// Mitsubishi GX Developer project: 12-202_201204121600   PLC: FX3U

PROGRAM MAIN
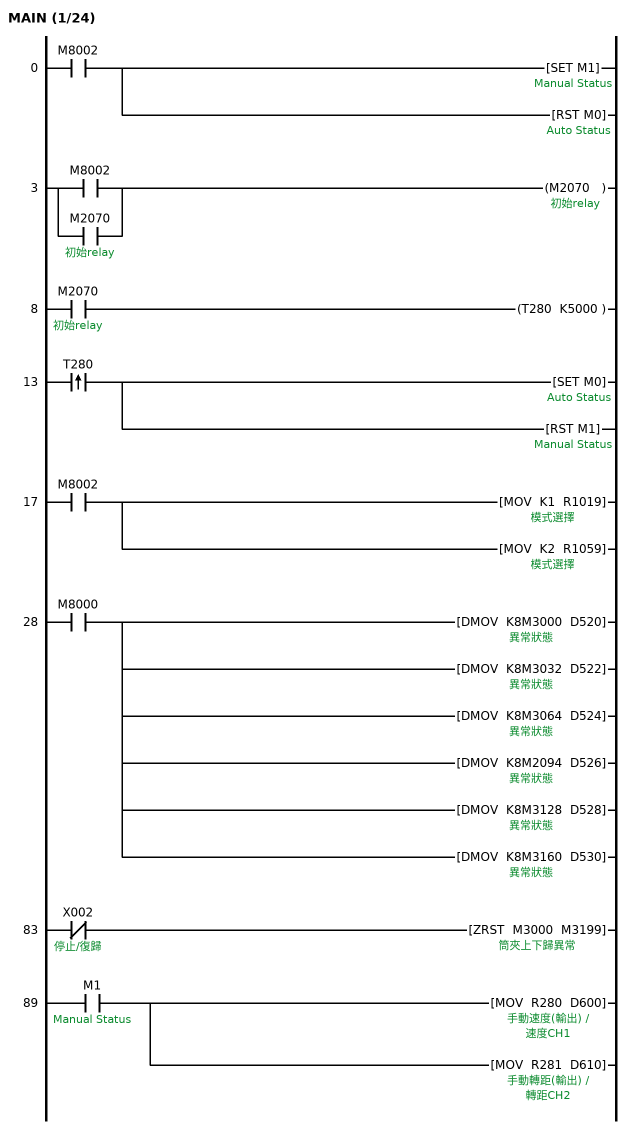
0     LD      M8002
      SET     M1  ; Manual Status
      RST     M0  ; Auto Status
3     LD      M8002
      OR      M2070  ; 初始relay
      OUT     M2070  ; 初始relay
8     LD      M2070  ; 初始relay
      OUT     T280 K5000
13    LDP     T280
      SET     M0  ; Auto Status
      RST     M1  ; Manual Status
17    LD      M8002
      MOV     K1 R1019  ; 模式選擇
      MOV     K2 R1059  ; 模式選擇
28    LD      M8000
      DMOV    K8M3000 D520  ; 筒夾上下歸異常 / 異常狀態
      DMOV    K8M3032 D522  ; 異常狀態
      DMOV    K8M3064 D524  ; 異常狀態
      DMOV    K8M2094 D526  ; 異常狀態
      DMOV    K8M3128 D528  ; 異常狀態
      DMOV    K8M3160 D530  ; 異常狀態
83    LDI     X002  ; 停止/復歸
      ZRST    M3000 M3199
89    LD      M1  ; Manual Status
      MOV     R280 D600  ; 手動速度(輸出) / 速度CH1
      MOV     R281 D610  ; 手動轉距(輸出) / 轉距CH2
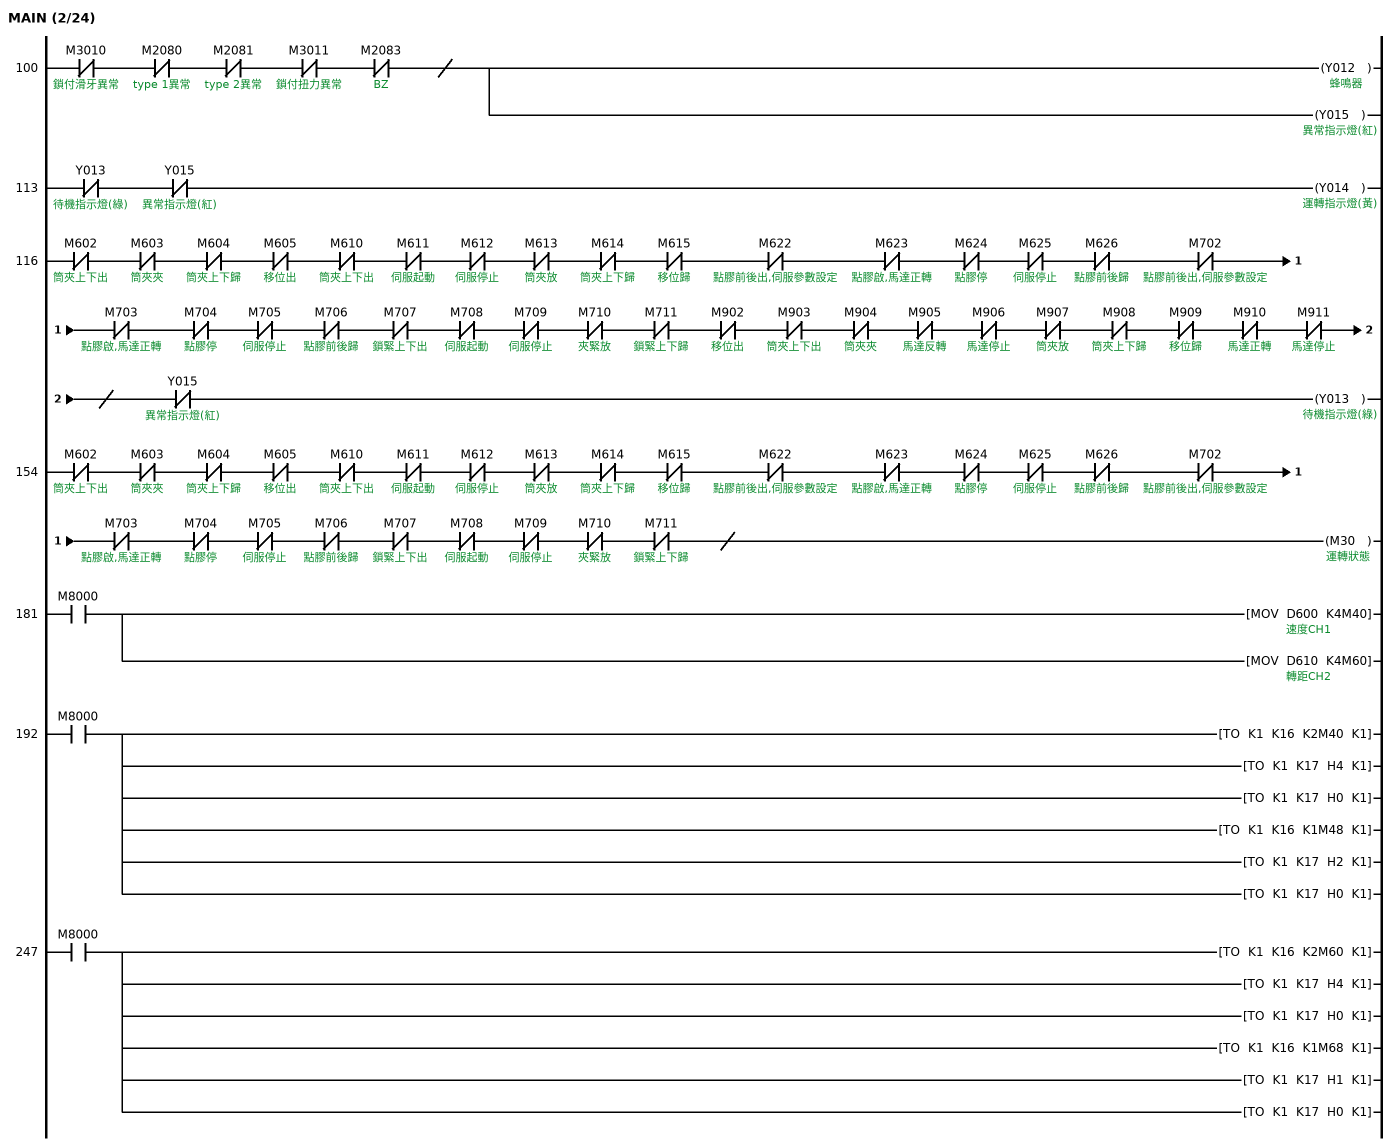
100   LDI     M3010  ; 鎖付滑牙異常
      ANI     M2080  ; type 1異常
      ANI     M2081  ; type 2異常
      ANI     M3011  ; 鎖付扭力異常
      ANI     M2083  ; BZ
      INV
      OUT     Y012  ; 蜂鳴器
      OUT     Y015  ; 異常指示燈(紅)
113   LDI     Y013  ; 待機指示燈(綠)
      ANI     Y015  ; 異常指示燈(紅)
      OUT     Y014  ; 運轉指示燈(黃)
116   LDI     M602  ; 筒夾上下出
      ANI     M603  ; 筒夾夾
      ANI     M604  ; 筒夾上下歸
      ANI     M605  ; 移位出
      ANI     M610  ; 筒夾上下出
      ANI     M611  ; 伺服起動
      ANI     M612  ; 伺服停止
      ANI     M613  ; 筒夾放
      ANI     M614  ; 筒夾上下歸
      ANI     M615  ; 移位歸
      ANI     M622  ; 點膠前後出,伺服參數設定
      ANI     M623  ; 點膠啟,馬達正轉
      ANI     M624  ; 點膠停
      ANI     M625  ; 伺服停止
      ANI     M626  ; 點膠前後歸
      ANI     M702  ; 點膠前後出,伺服參數設定
      ANI     M703  ; 點膠啟,馬達正轉
      ANI     M704  ; 點膠停
      ANI     M705  ; 伺服停止
      ANI     M706  ; 點膠前後歸
      ANI     M707  ; 鎖緊上下出
      ANI     M708  ; 伺服起動
      ANI     M709  ; 伺服停止
      ANI     M710  ; 夾緊放
      ANI     M711  ; 鎖緊上下歸
      ANI     M902  ; 移位出
      ANI     M903  ; 筒夾上下出
      ANI     M904  ; 筒夾夾
      ANI     M905  ; 馬達反轉
      ANI     M906  ; 馬達停止
      ANI     M907  ; 筒夾放
      ANI     M908  ; 筒夾上下歸
      ANI     M909  ; 移位歸
      ANI     M910  ; 馬達正轉
      ANI     M911  ; 馬達停止
      INV
      ANI     Y015  ; 異常指示燈(紅)
      OUT     Y013  ; 待機指示燈(綠)
154   LDI     M602  ; 筒夾上下出
      ANI     M603  ; 筒夾夾
      ANI     M604  ; 筒夾上下歸
      ANI     M605  ; 移位出
      ANI     M610  ; 筒夾上下出
      ANI     M611  ; 伺服起動
      ANI     M612  ; 伺服停止
      ANI     M613  ; 筒夾放
      ANI     M614  ; 筒夾上下歸
      ANI     M615  ; 移位歸
      ANI     M622  ; 點膠前後出,伺服參數設定
      ANI     M623  ; 點膠啟,馬達正轉
      ANI     M624  ; 點膠停
      ANI     M625  ; 伺服停止
      ANI     M626  ; 點膠前後歸
      ANI     M702  ; 點膠前後出,伺服參數設定
      ANI     M703  ; 點膠啟,馬達正轉
      ANI     M704  ; 點膠停
      ANI     M705  ; 伺服停止
      ANI     M706  ; 點膠前後歸
      ANI     M707  ; 鎖緊上下出
      ANI     M708  ; 伺服起動
      ANI     M709  ; 伺服停止
      ANI     M710  ; 夾緊放
      ANI     M711  ; 鎖緊上下歸
      INV
      OUT     M30  ; 運轉狀態
181   LD      M8000
      MOV     D600 K4M40  ; DA用
      MOV     D610 K4M60  ; DA用
192   LD      M8000
      TO      K1 K16 K2M40 K1
      TO      K1 K17 H4 K1
      TO      K1 K17 H0 K1
      TO      K1 K16 K1M48 K1  ; DA用
      TO      K1 K17 H2 K1
      TO      K1 K17 H0 K1
247   LD      M8000
      TO      K1 K16 K2M60 K1
      TO      K1 K17 H4 K1
      TO      K1 K17 H0 K1
      TO      K1 K16 K1M68 K1  ; DA用
      TO      K1 K17 H1 K1
      TO      K1 K17 H0 K1
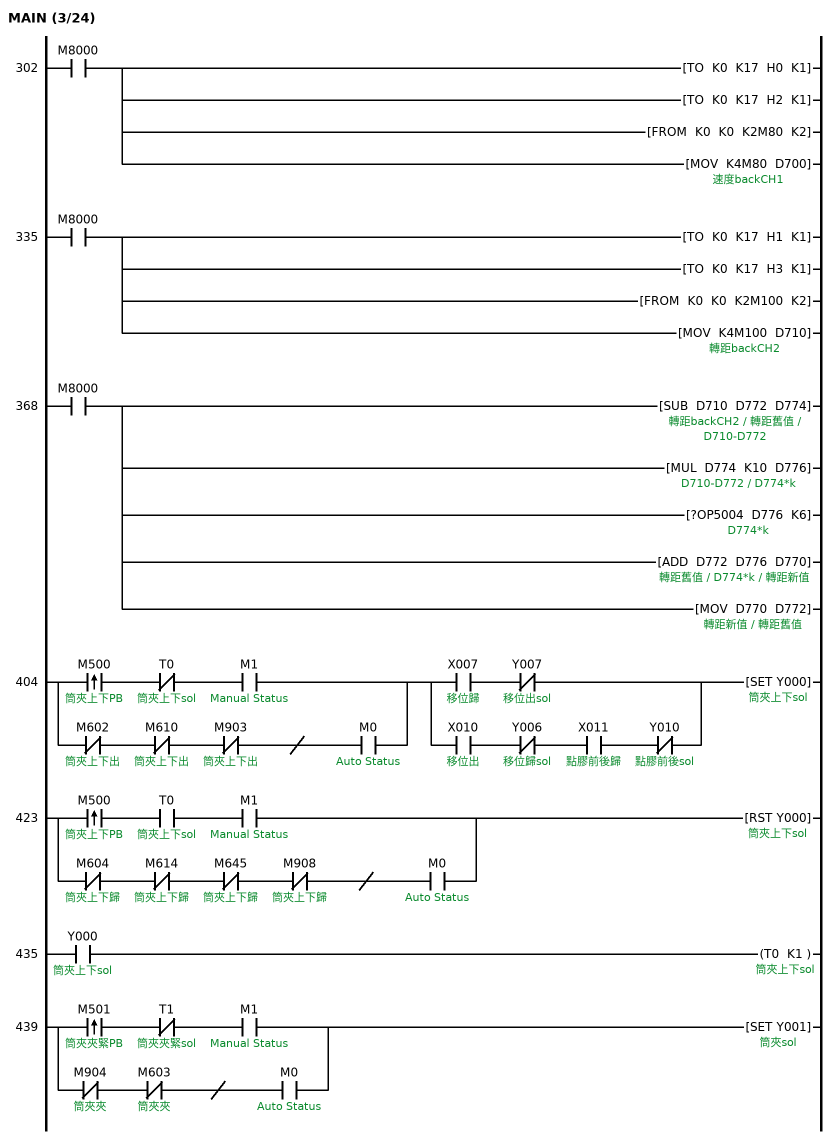
302   LD      M8000
      TO      K0 K17 H0 K1
      TO      K0 K17 H2 K1
      FROM    K0 K0 K2M80 K2  ; AD用
      MOV     K4M80 D700  ; 速度backCH1
335   LD      M8000
      TO      K0 K17 H1 K1
      TO      K0 K17 H3 K1
      FROM    K0 K0 K2M100 K2  ; AD用
      MOV     K4M100 D710  ; 轉距backCH2
368   LD      M8000
      SUB     D710 D772 D774  ; 轉距舊值 / D710-D772
      MUL     D774 K10 D776  ; D774*k
      ?OP5004 D776 K6
      ADD     D772 D776 D770  ; 轉距新值
      MOV     D770 D772
404   LDP     M500  ; 筒夾上下PB
      ANI     T0  ; 筒夾上下sol
      AND     M1  ; Manual Status
      LDI     M602  ; 筒夾上下出
      ANI     M610  ; 筒夾上下出
      ANI     M903  ; 筒夾上下出
      INV
      AND     M0  ; Auto Status
      ORB
      LD      X007  ; 移位歸
      ANI     Y007  ; 移位出sol
      LD      X010  ; 移位出
      ANI     Y006  ; 移位歸sol
      AND     X011  ; 點膠前後歸
      ANI     Y010  ; 點膠前後sol
      ORB
      ANB
      SET     Y000  ; 筒夾上下sol
423   LDP     M500  ; 筒夾上下PB
      AND     T0  ; 筒夾上下sol
      AND     M1  ; Manual Status
      LDI     M604  ; 筒夾上下歸
      ANI     M614  ; 筒夾上下歸
      ANI     M645  ; 筒夾上下歸
      ANI     M908  ; 筒夾上下歸
      INV
      AND     M0  ; Auto Status
      ORB
      RST     Y000  ; 筒夾上下sol
435   LD      Y000  ; 筒夾上下sol
      OUT     T0 K1  ; 筒夾上下sol
439   LDP     M501  ; 筒夾夾緊PB
      ANI     T1  ; 筒夾夾緊sol
      AND     M1  ; Manual Status
      LDI     M904  ; 筒夾夾
      ANI     M603  ; 筒夾夾
      INV
      AND     M0  ; Auto Status
      ORB
      SET     Y001  ; 筒夾sol
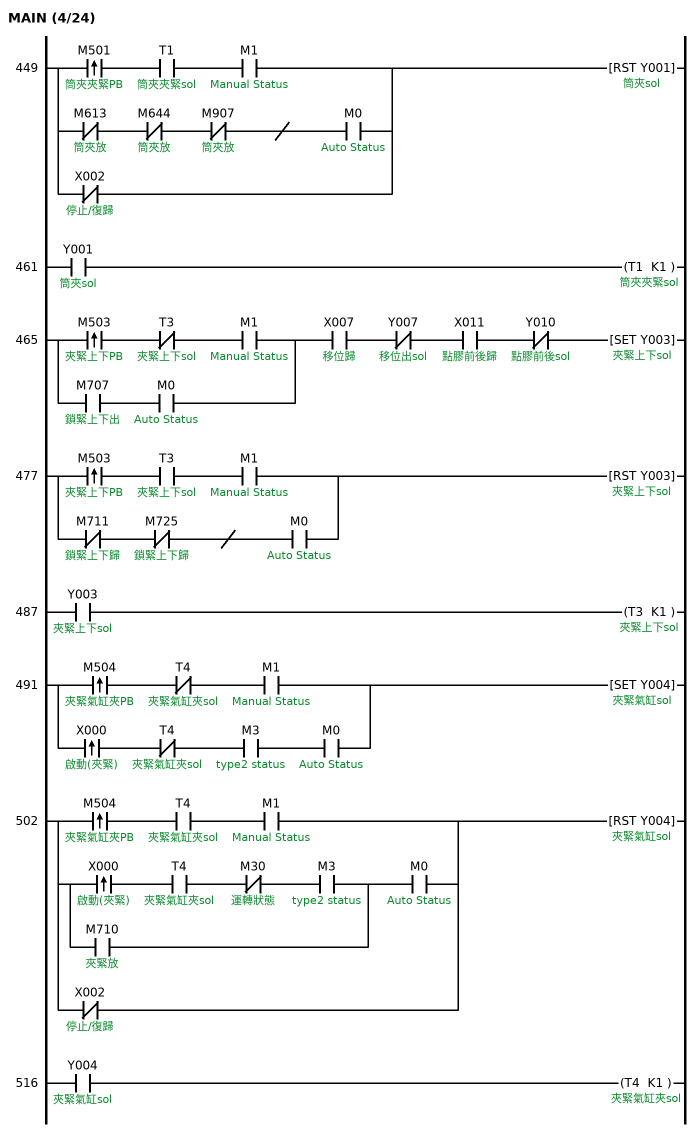
449   LDP     M501  ; 筒夾夾緊PB
      AND     T1  ; 筒夾夾緊sol
      AND     M1  ; Manual Status
      LDI     M613  ; 筒夾放
      ANI     M644  ; 筒夾放
      ANI     M907  ; 筒夾放
      INV
      AND     M0  ; Auto Status
      ORB
      ORI     X002  ; 停止/復歸
      RST     Y001  ; 筒夾sol
461   LD      Y001  ; 筒夾sol
      OUT     T1 K1  ; 筒夾夾緊sol
465   LDP     M503  ; 夾緊上下PB
      ANI     T3  ; 夾緊上下sol
      AND     M1  ; Manual Status
      LD      M707  ; 鎖緊上下出
      AND     M0  ; Auto Status
      ORB
      AND     X007  ; 移位歸
      ANI     Y007  ; 移位出sol
      AND     X011  ; 點膠前後歸
      ANI     Y010  ; 點膠前後sol
      SET     Y003  ; 夾緊上下sol
477   LDP     M503  ; 夾緊上下PB
      AND     T3  ; 夾緊上下sol
      AND     M1  ; Manual Status
      LDI     M711  ; 鎖緊上下歸
      ANI     M725  ; 鎖緊上下歸
      INV
      AND     M0  ; Auto Status
      ORB
      RST     Y003  ; 夾緊上下sol
487   LD      Y003  ; 夾緊上下sol
      OUT     T3 K1  ; 夾緊上下sol
491   LDP     M504  ; 夾緊氣缸夾PB
      ANI     T4  ; 夾緊氣缸夾sol
      AND     M1  ; Manual Status
      LDP     X000  ; 啟動(夾緊)
      ANI     T4  ; 夾緊氣缸夾sol
      AND     M3  ; type2 status
      AND     M0  ; Auto Status
      ORB
      SET     Y004  ; 夾緊氣缸sol
502   LDP     M504  ; 夾緊氣缸夾PB
      AND     T4  ; 夾緊氣缸夾sol
      AND     M1  ; Manual Status
      LDP     X000  ; 啟動(夾緊)
      AND     T4  ; 夾緊氣缸夾sol
      ANI     M30  ; 運轉狀態
      AND     M3  ; type2 status
      OR      M710  ; 夾緊放
      AND     M0  ; Auto Status
      ORB
      ORI     X002  ; 停止/復歸
      RST     Y004  ; 夾緊氣缸sol
516   LD      Y004  ; 夾緊氣缸sol
      OUT     T4 K1  ; 夾緊氣缸夾sol
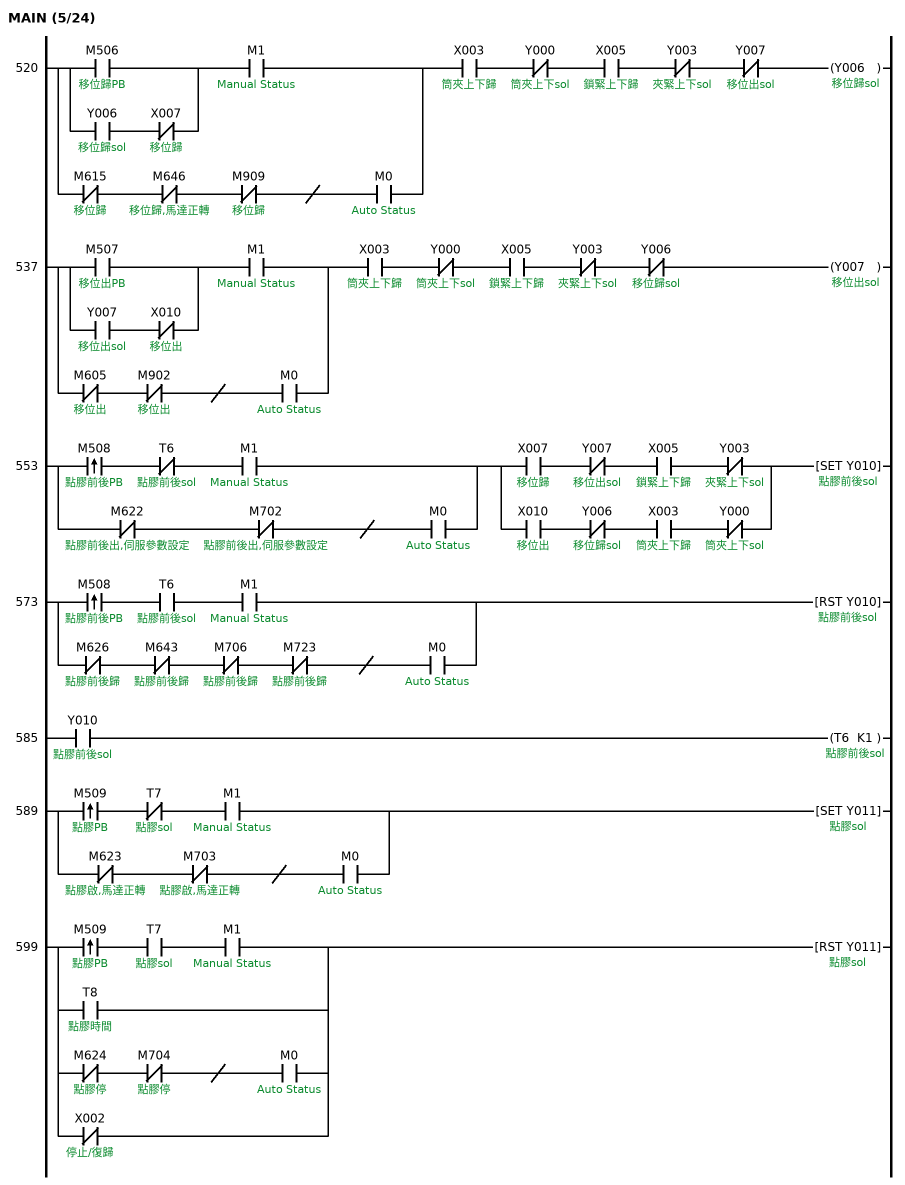
520   LD      M506  ; 移位歸PB
      LD      Y006  ; 移位歸sol
      ANI     X007  ; 移位歸
      ORB
      AND     M1  ; Manual Status
      LDI     M615  ; 移位歸
      ANI     M646  ; 移位歸,馬達正轉
      ANI     M909  ; 移位歸
      INV
      AND     M0  ; Auto Status
      ORB
      AND     X003  ; 筒夾上下歸
      ANI     Y000  ; 筒夾上下sol
      AND     X005  ; 鎖緊上下歸
      ANI     Y003  ; 夾緊上下sol
      ANI     Y007  ; 移位出sol
      OUT     Y006  ; 移位歸sol
537   LD      M507  ; 移位出PB
      LD      Y007  ; 移位出sol
      ANI     X010  ; 移位出
      ORB
      AND     M1  ; Manual Status
      LDI     M605  ; 移位出
      ANI     M902  ; 移位出
      INV
      AND     M0  ; Auto Status
      ORB
      AND     X003  ; 筒夾上下歸
      ANI     Y000  ; 筒夾上下sol
      AND     X005  ; 鎖緊上下歸
      ANI     Y003  ; 夾緊上下sol
      ANI     Y006  ; 移位歸sol
      OUT     Y007  ; 移位出sol
553   LDP     M508  ; 點膠前後PB
      ANI     T6  ; 點膠前後sol
      AND     M1  ; Manual Status
      LDI     M622  ; 點膠前後出,伺服參數設定
      ANI     M702  ; 點膠前後出,伺服參數設定
      INV
      AND     M0  ; Auto Status
      ORB
      LD      X007  ; 移位歸
      ANI     Y007  ; 移位出sol
      AND     X005  ; 鎖緊上下歸
      ANI     Y003  ; 夾緊上下sol
      LD      X010  ; 移位出
      ANI     Y006  ; 移位歸sol
      AND     X003  ; 筒夾上下歸
      ANI     Y000  ; 筒夾上下sol
      ORB
      ANB
      SET     Y010  ; 點膠前後sol
573   LDP     M508  ; 點膠前後PB
      AND     T6  ; 點膠前後sol
      AND     M1  ; Manual Status
      LDI     M626  ; 點膠前後歸
      ANI     M643  ; 點膠前後歸
      ANI     M706  ; 點膠前後歸
      ANI     M723  ; 點膠前後歸
      INV
      AND     M0  ; Auto Status
      ORB
      RST     Y010  ; 點膠前後sol
585   LD      Y010  ; 點膠前後sol
      OUT     T6 K1  ; 點膠前後sol
589   LDP     M509  ; 點膠PB
      ANI     T7  ; 點膠sol
      AND     M1  ; Manual Status
      LDI     M623  ; 點膠啟,馬達正轉
      ANI     M703  ; 點膠啟,馬達正轉
      INV
      AND     M0  ; Auto Status
      ORB
      SET     Y011  ; 點膠sol
599   LDP     M509  ; 點膠PB
      AND     T7  ; 點膠sol
      AND     M1  ; Manual Status
      OR      T8  ; 點膠時間
      LDI     M624  ; 點膠停
      ANI     M704  ; 點膠停
      INV
      AND     M0  ; Auto Status
      ORB
      ORI     X002  ; 停止/復歸
      RST     Y011  ; 點膠sol
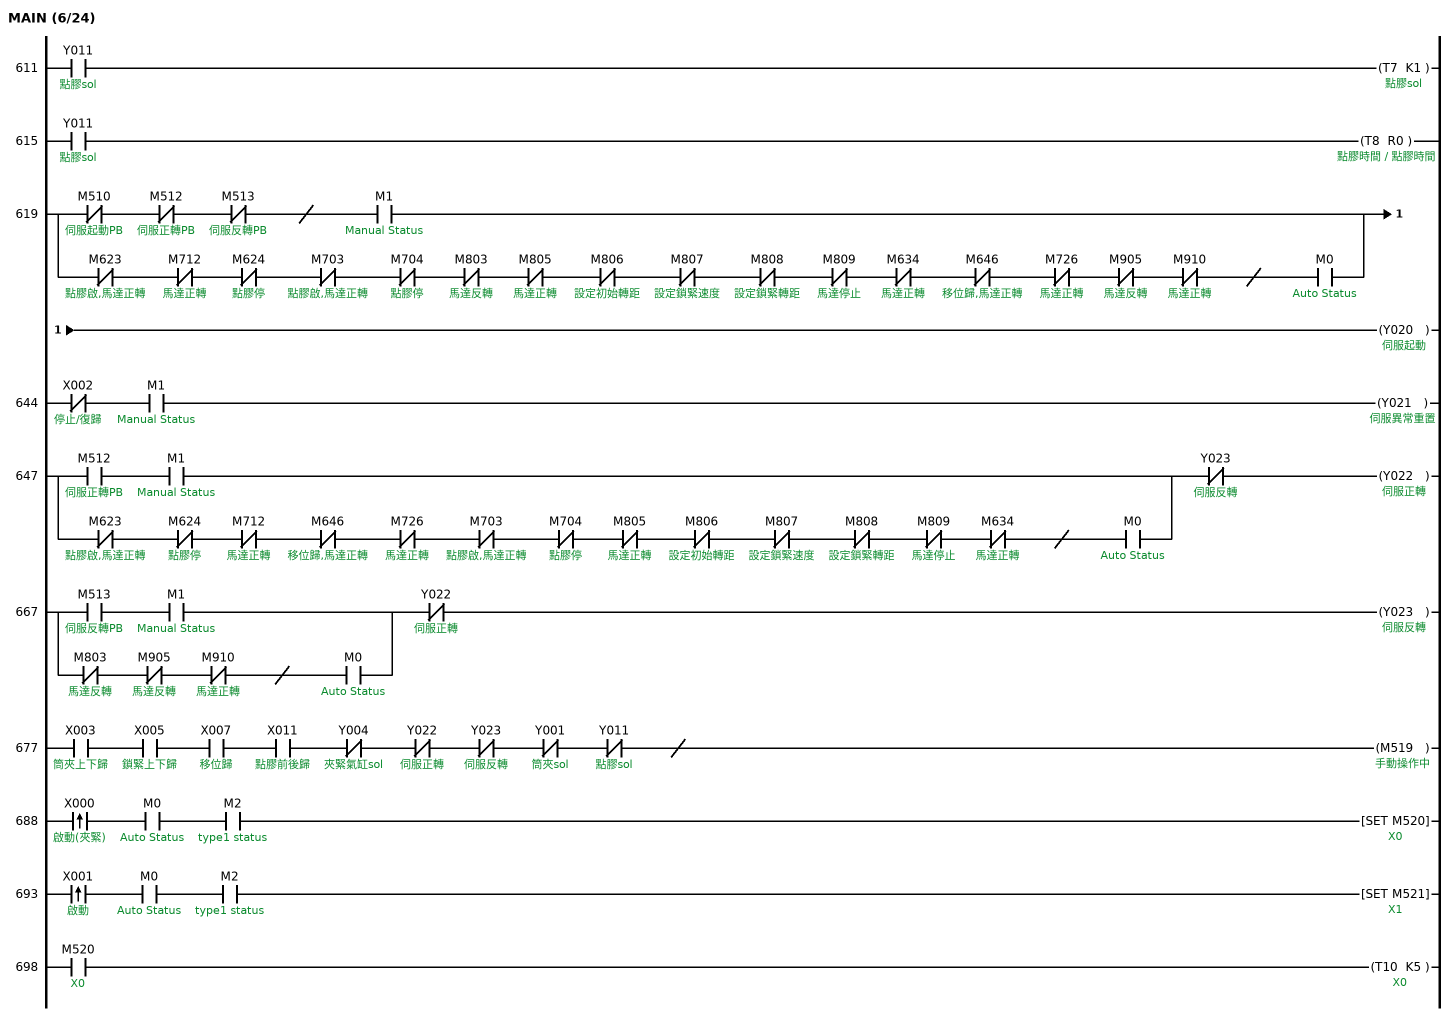
611   LD      Y011  ; 點膠sol
      OUT     T7 K1  ; 點膠sol
615   LD      Y011  ; 點膠sol
      OUT     T8 R0  ; 點膠時間 / 點膠時間
619   LDI     M510  ; 伺服起動PB
      ANI     M512  ; 伺服正轉PB
      ANI     M513  ; 伺服反轉PB
      INV
      AND     M1  ; Manual Status
      LDI     M623  ; 點膠啟,馬達正轉
      ANI     M712  ; 馬達正轉
      ANI     M624  ; 點膠停
      ANI     M703  ; 點膠啟,馬達正轉
      ANI     M704  ; 點膠停
      ANI     M803  ; 馬達反轉
      ANI     M805  ; 馬達正轉
      ANI     M806  ; 設定初始轉距
      ANI     M807  ; 設定鎖緊速度
      ANI     M808  ; 設定鎖緊轉距
      ANI     M809  ; 馬達停止
      ANI     M634  ; 馬達正轉
      ANI     M646  ; 移位歸,馬達正轉
      ANI     M726  ; 馬達正轉
      ANI     M905  ; 馬達反轉
      ANI     M910  ; 馬達正轉
      INV
      AND     M0  ; Auto Status
      ORB
      OUT     Y020  ; 伺服起動
644   LDI     X002  ; 停止/復歸
      AND     M1  ; Manual Status
      OUT     Y021  ; 伺服異常重置
647   LD      M512  ; 伺服正轉PB
      AND     M1  ; Manual Status
      LDI     M623  ; 點膠啟,馬達正轉
      ANI     M624  ; 點膠停
      ANI     M712  ; 馬達正轉
      ANI     M646  ; 移位歸,馬達正轉
      ANI     M726  ; 馬達正轉
      ANI     M703  ; 點膠啟,馬達正轉
      ANI     M704  ; 點膠停
      ANI     M805  ; 馬達正轉
      ANI     M806  ; 設定初始轉距
      ANI     M807  ; 設定鎖緊速度
      ANI     M808  ; 設定鎖緊轉距
      ANI     M809  ; 馬達停止
      ANI     M634  ; 馬達正轉
      INV
      AND     M0  ; Auto Status
      ORB
      ANI     Y023  ; 伺服反轉
      OUT     Y022  ; 伺服正轉
667   LD      M513  ; 伺服反轉PB
      AND     M1  ; Manual Status
      LDI     M803  ; 馬達反轉
      ANI     M905  ; 馬達反轉
      ANI     M910  ; 馬達正轉
      INV
      AND     M0  ; Auto Status
      ORB
      ANI     Y022  ; 伺服正轉
      OUT     Y023  ; 伺服反轉
677   LD      X003  ; 筒夾上下歸
      AND     X005  ; 鎖緊上下歸
      AND     X007  ; 移位歸
      AND     X011  ; 點膠前後歸
      ANI     Y004  ; 夾緊氣缸sol
      ANI     Y022  ; 伺服正轉
      ANI     Y023  ; 伺服反轉
      ANI     Y001  ; 筒夾sol
      ANI     Y011  ; 點膠sol
      INV
      OUT     M519  ; 手動操作中
688   LDP     X000  ; 啟動(夾緊)
      AND     M0  ; Auto Status
      AND     M2  ; type1 status
      SET     M520  ; X0
693   LDP     X001  ; 啟動
      AND     M0  ; Auto Status
      AND     M2  ; type1 status
      SET     M521  ; X1
698   LD      M520  ; X0
      OUT     T10 K5  ; X0
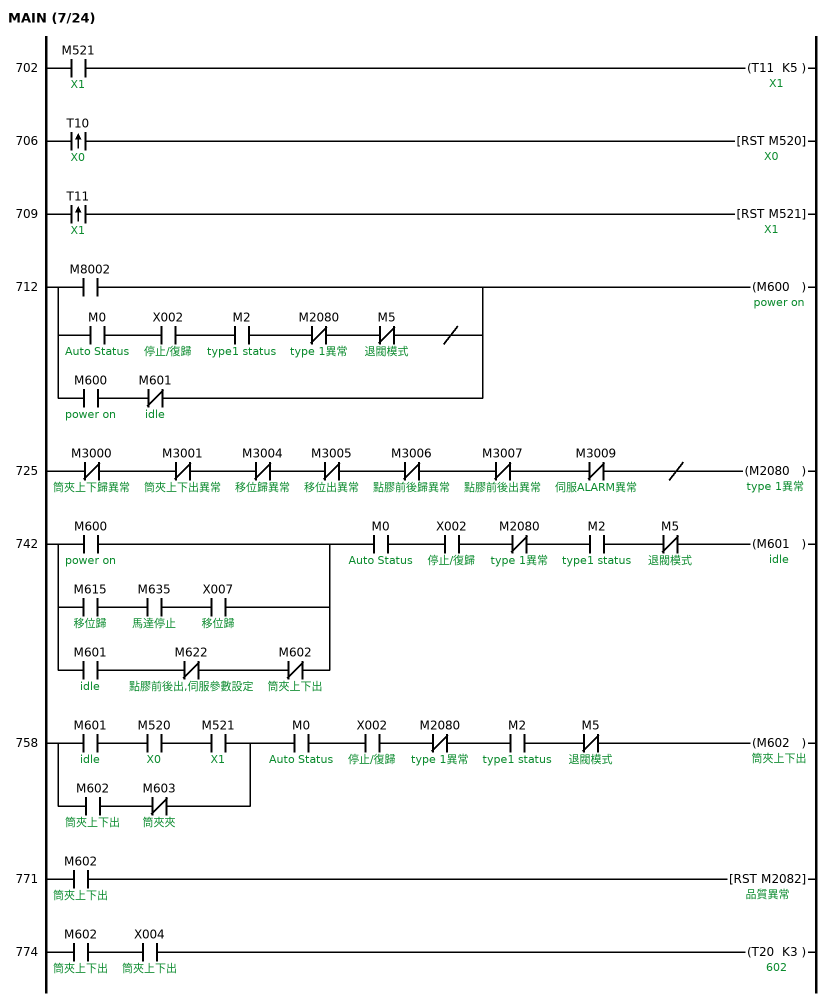
702   LD      M521  ; X1
      OUT     T11 K5  ; X1
706   LDP     T10  ; X0
      RST     M520  ; X0
709   LDP     T11  ; X1
      RST     M521  ; X1
712   LD      M8002
      LD      M0  ; Auto Status
      AND     X002  ; 停止/復歸
      AND     M2  ; type1 status
      ANI     M2080  ; type 1異常
      ANI     M5  ; 退閥模式
      INV
      ORB
      LD      M600  ; power on
      ANI     M601  ; idle
      ORB
      OUT     M600  ; power on
725   LDI     M3000  ; 筒夾上下歸異常
      ANI     M3001  ; 筒夾上下出異常
      ANI     M3004  ; 移位歸異常
      ANI     M3005  ; 移位出異常
      ANI     M3006  ; 點膠前後歸異常
      ANI     M3007  ; 點膠前後出異常
      ANI     M3009  ; 伺服ALARM異常
      INV
      OUT     M2080  ; type 1異常
742   LD      M600  ; power on
      LD      M615  ; 移位歸
      AND     M635  ; 馬達停止
      AND     X007  ; 移位歸
      ORB
      LD      M601  ; idle
      ANI     M622  ; 點膠前後出,伺服參數設定
      ANI     M602  ; 筒夾上下出
      ORB
      AND     M0  ; Auto Status
      AND     X002  ; 停止/復歸
      ANI     M2080  ; type 1異常
      AND     M2  ; type1 status
      ANI     M5  ; 退閥模式
      OUT     M601  ; idle
758   LD      M601  ; idle
      AND     M520  ; X0
      AND     M521  ; X1
      LD      M602  ; 筒夾上下出
      ANI     M603  ; 筒夾夾
      ORB
      AND     M0  ; Auto Status
      AND     X002  ; 停止/復歸
      ANI     M2080  ; type 1異常
      AND     M2  ; type1 status
      ANI     M5  ; 退閥模式
      OUT     M602  ; 筒夾上下出
771   LD      M602  ; 筒夾上下出
      RST     M2082  ; 品質異常
774   LD      M602  ; 筒夾上下出
      AND     X004  ; 筒夾上下出
      OUT     T20 K3  ; 602
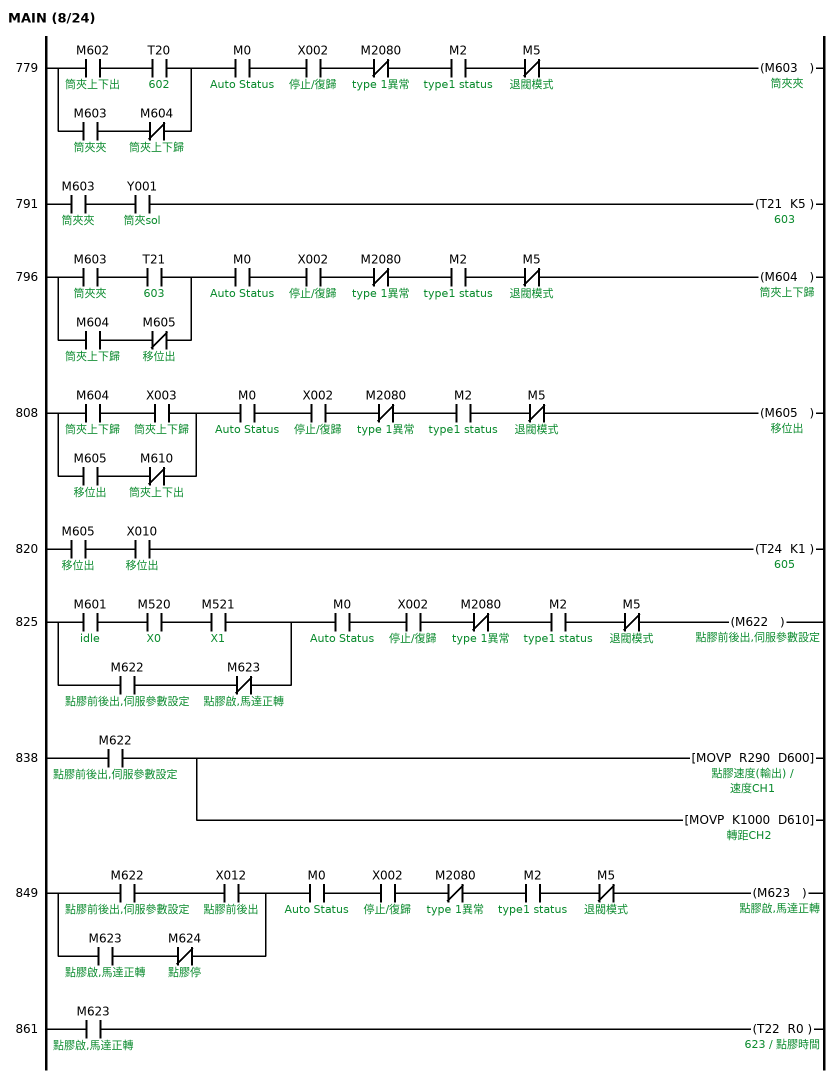
779   LD      M602  ; 筒夾上下出
      AND     T20  ; 602
      LD      M603  ; 筒夾夾
      ANI     M604  ; 筒夾上下歸
      ORB
      AND     M0  ; Auto Status
      AND     X002  ; 停止/復歸
      ANI     M2080  ; type 1異常
      AND     M2  ; type1 status
      ANI     M5  ; 退閥模式
      OUT     M603  ; 筒夾夾
791   LD      M603  ; 筒夾夾
      AND     Y001  ; 筒夾sol
      OUT     T21 K5  ; 603
796   LD      M603  ; 筒夾夾
      AND     T21  ; 603
      LD      M604  ; 筒夾上下歸
      ANI     M605  ; 移位出
      ORB
      AND     M0  ; Auto Status
      AND     X002  ; 停止/復歸
      ANI     M2080  ; type 1異常
      AND     M2  ; type1 status
      ANI     M5  ; 退閥模式
      OUT     M604  ; 筒夾上下歸
808   LD      M604  ; 筒夾上下歸
      AND     X003  ; 筒夾上下歸
      LD      M605  ; 移位出
      ANI     M610  ; 筒夾上下出
      ORB
      AND     M0  ; Auto Status
      AND     X002  ; 停止/復歸
      ANI     M2080  ; type 1異常
      AND     M2  ; type1 status
      ANI     M5  ; 退閥模式
      OUT     M605  ; 移位出
820   LD      M605  ; 移位出
      AND     X010  ; 移位出
      OUT     T24 K1  ; 605
825   LD      M601  ; idle
      AND     M520  ; X0
      AND     M521  ; X1
      LD      M622  ; 點膠前後出,伺服參數設定
      ANI     M623  ; 點膠啟,馬達正轉
      ORB
      AND     M0  ; Auto Status
      AND     X002  ; 停止/復歸
      ANI     M2080  ; type 1異常
      AND     M2  ; type1 status
      ANI     M5  ; 退閥模式
      OUT     M622  ; 點膠前後出,伺服參數設定
838   LD      M622  ; 點膠前後出,伺服參數設定
      MOVP    R290 D600  ; 點膠速度(輸出)
      MOVP    K1000 D610
849   LD      M622  ; 點膠前後出,伺服參數設定
      AND     X012  ; 點膠前後出
      LD      M623  ; 點膠啟,馬達正轉
      ANI     M624  ; 點膠停
      ORB
      AND     M0  ; Auto Status
      AND     X002  ; 停止/復歸
      ANI     M2080  ; type 1異常
      AND     M2  ; type1 status
      ANI     M5  ; 退閥模式
      OUT     M623  ; 點膠啟,馬達正轉
861   LD      M623  ; 點膠啟,馬達正轉
      OUT     T22 R0  ; 623 / 點膠時間
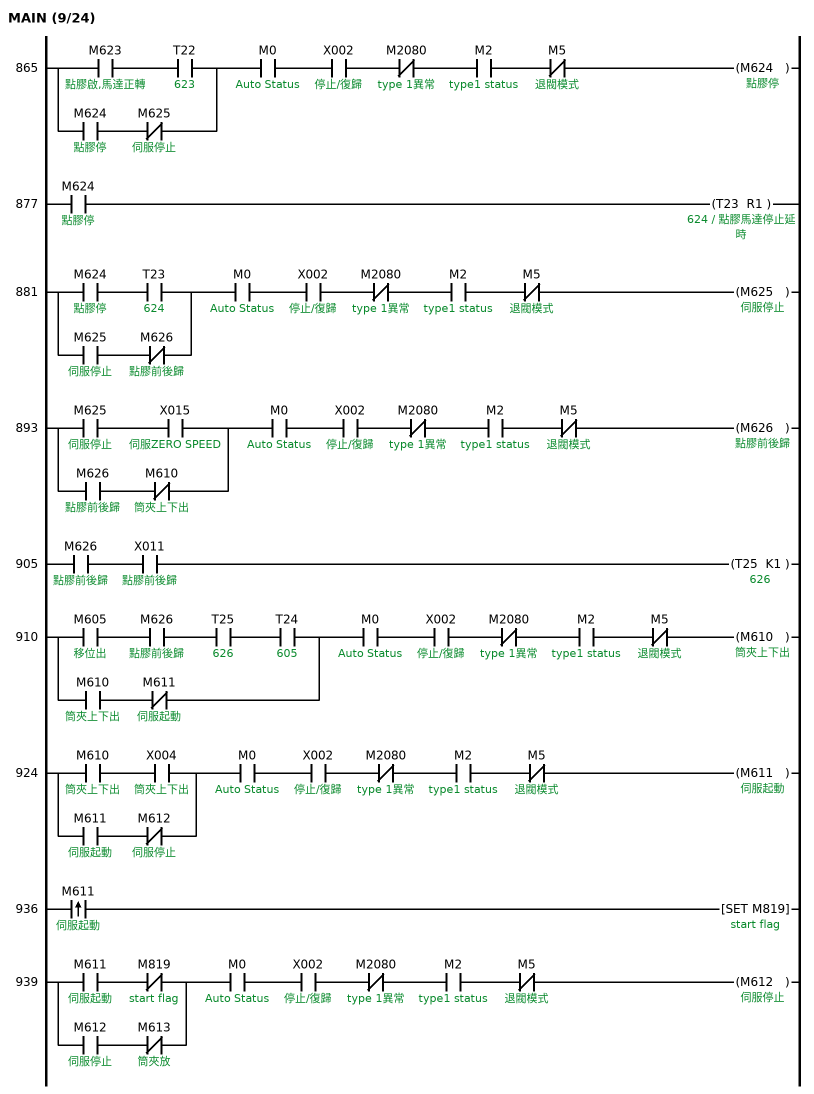
865   LD      M623  ; 點膠啟,馬達正轉
      AND     T22  ; 623
      LD      M624  ; 點膠停
      ANI     M625  ; 伺服停止
      ORB
      AND     M0  ; Auto Status
      AND     X002  ; 停止/復歸
      ANI     M2080  ; type 1異常
      AND     M2  ; type1 status
      ANI     M5  ; 退閥模式
      OUT     M624  ; 點膠停
877   LD      M624  ; 點膠停
      OUT     T23 R1  ; 624 / 點膠馬達停止延時
881   LD      M624  ; 點膠停
      AND     T23  ; 624
      LD      M625  ; 伺服停止
      ANI     M626  ; 點膠前後歸
      ORB
      AND     M0  ; Auto Status
      AND     X002  ; 停止/復歸
      ANI     M2080  ; type 1異常
      AND     M2  ; type1 status
      ANI     M5  ; 退閥模式
      OUT     M625  ; 伺服停止
893   LD      M625  ; 伺服停止
      AND     X015  ; 伺服ZERO SPEED
      LD      M626  ; 點膠前後歸
      ANI     M610  ; 筒夾上下出
      ORB
      AND     M0  ; Auto Status
      AND     X002  ; 停止/復歸
      ANI     M2080  ; type 1異常
      AND     M2  ; type1 status
      ANI     M5  ; 退閥模式
      OUT     M626  ; 點膠前後歸
905   LD      M626  ; 點膠前後歸
      AND     X011  ; 點膠前後歸
      OUT     T25 K1  ; 626
910   LD      M605  ; 移位出
      AND     M626  ; 點膠前後歸
      AND     T25  ; 626
      AND     T24  ; 605
      LD      M610  ; 筒夾上下出
      ANI     M611  ; 伺服起動
      ORB
      AND     M0  ; Auto Status
      AND     X002  ; 停止/復歸
      ANI     M2080  ; type 1異常
      AND     M2  ; type1 status
      ANI     M5  ; 退閥模式
      OUT     M610  ; 筒夾上下出
924   LD      M610  ; 筒夾上下出
      AND     X004  ; 筒夾上下出
      LD      M611  ; 伺服起動
      ANI     M612  ; 伺服停止
      ORB
      AND     M0  ; Auto Status
      AND     X002  ; 停止/復歸
      ANI     M2080  ; type 1異常
      AND     M2  ; type1 status
      ANI     M5  ; 退閥模式
      OUT     M611  ; 伺服起動
936   LDP     M611  ; 伺服起動
      SET     M819  ; start flag
939   LD      M611  ; 伺服起動
      ANI     M819  ; start flag
      LD      M612  ; 伺服停止
      ANI     M613  ; 筒夾放
      ORB
      AND     M0  ; Auto Status
      AND     X002  ; 停止/復歸
      ANI     M2080  ; type 1異常
      AND     M2  ; type1 status
      ANI     M5  ; 退閥模式
      OUT     M612  ; 伺服停止
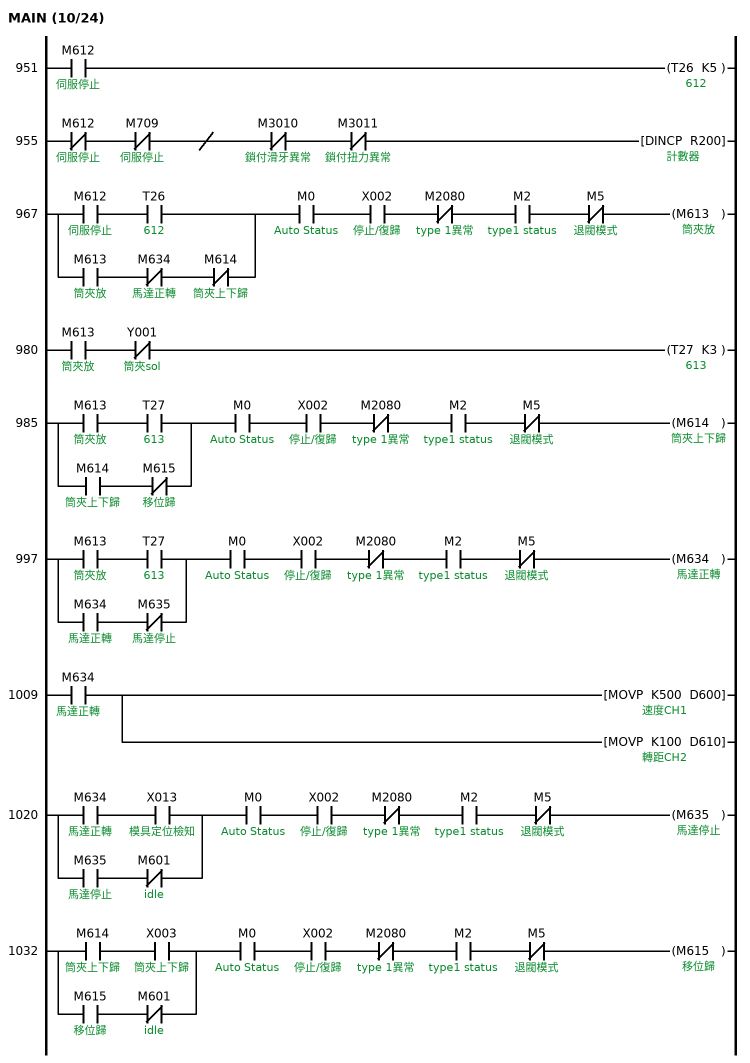
951   LD      M612  ; 伺服停止
      OUT     T26 K5  ; 612
955   LDI     M612  ; 伺服停止
      ANI     M709  ; 伺服停止
      INV
      ANI     M3010  ; 鎖付滑牙異常
      ANI     M3011  ; 鎖付扭力異常
      DINCP   R200  ; 計數器
967   LD      M612  ; 伺服停止
      AND     T26  ; 612
      LD      M613  ; 筒夾放
      ANI     M634  ; 馬達正轉
      ANI     M614  ; 筒夾上下歸
      ORB
      AND     M0  ; Auto Status
      AND     X002  ; 停止/復歸
      ANI     M2080  ; type 1異常
      AND     M2  ; type1 status
      ANI     M5  ; 退閥模式
      OUT     M613  ; 筒夾放
980   LD      M613  ; 筒夾放
      ANI     Y001  ; 筒夾sol
      OUT     T27 K3  ; 613
985   LD      M613  ; 筒夾放
      AND     T27  ; 613
      LD      M614  ; 筒夾上下歸
      ANI     M615  ; 移位歸
      ORB
      AND     M0  ; Auto Status
      AND     X002  ; 停止/復歸
      ANI     M2080  ; type 1異常
      AND     M2  ; type1 status
      ANI     M5  ; 退閥模式
      OUT     M614  ; 筒夾上下歸
997   LD      M613  ; 筒夾放
      AND     T27  ; 613
      LD      M634  ; 馬達正轉
      ANI     M635  ; 馬達停止
      ORB
      AND     M0  ; Auto Status
      AND     X002  ; 停止/復歸
      ANI     M2080  ; type 1異常
      AND     M2  ; type1 status
      ANI     M5  ; 退閥模式
      OUT     M634  ; 馬達正轉
1009  LD      M634  ; 馬達正轉
      MOVP    K500 D600
      MOVP    K100 D610
1020  LD      M634  ; 馬達正轉
      AND     X013  ; 模具定位檢知
      LD      M635  ; 馬達停止
      ANI     M601  ; idle
      ORB
      AND     M0  ; Auto Status
      AND     X002  ; 停止/復歸
      ANI     M2080  ; type 1異常
      AND     M2  ; type1 status
      ANI     M5  ; 退閥模式
      OUT     M635  ; 馬達停止
1032  LD      M614  ; 筒夾上下歸
      AND     X003  ; 筒夾上下歸
      LD      M615  ; 移位歸
      ANI     M601  ; idle
      ORB
      AND     M0  ; Auto Status
      AND     X002  ; 停止/復歸
      ANI     M2080  ; type 1異常
      AND     M2  ; type1 status
      ANI     M5  ; 退閥模式
      OUT     M615  ; 移位歸
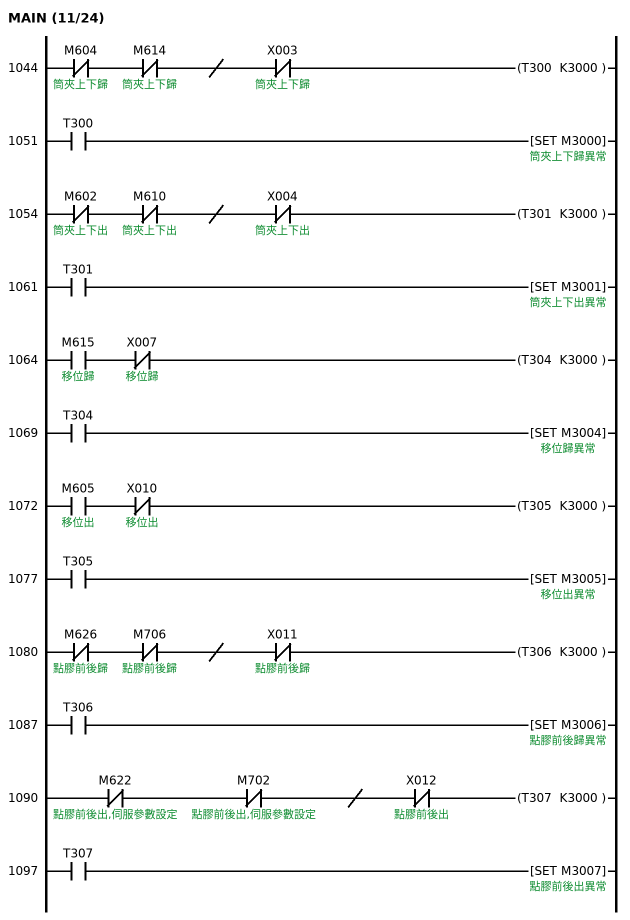
1044  LDI     M604  ; 筒夾上下歸
      ANI     M614  ; 筒夾上下歸
      INV
      ANI     X003  ; 筒夾上下歸
      OUT     T300 K3000
1051  LD      T300
      SET     M3000  ; 筒夾上下歸異常
1054  LDI     M602  ; 筒夾上下出
      ANI     M610  ; 筒夾上下出
      INV
      ANI     X004  ; 筒夾上下出
      OUT     T301 K3000
1061  LD      T301
      SET     M3001  ; 筒夾上下出異常
1064  LD      M615  ; 移位歸
      ANI     X007  ; 移位歸
      OUT     T304 K3000
1069  LD      T304
      SET     M3004  ; 移位歸異常
1072  LD      M605  ; 移位出
      ANI     X010  ; 移位出
      OUT     T305 K3000
1077  LD      T305
      SET     M3005  ; 移位出異常
1080  LDI     M626  ; 點膠前後歸
      ANI     M706  ; 點膠前後歸
      INV
      ANI     X011  ; 點膠前後歸
      OUT     T306 K3000
1087  LD      T306
      SET     M3006  ; 點膠前後歸異常
1090  LDI     M622  ; 點膠前後出,伺服參數設定
      ANI     M702  ; 點膠前後出,伺服參數設定
      INV
      ANI     X012  ; 點膠前後出
      OUT     T307 K3000
1097  LD      T307
      SET     M3007  ; 點膠前後出異常
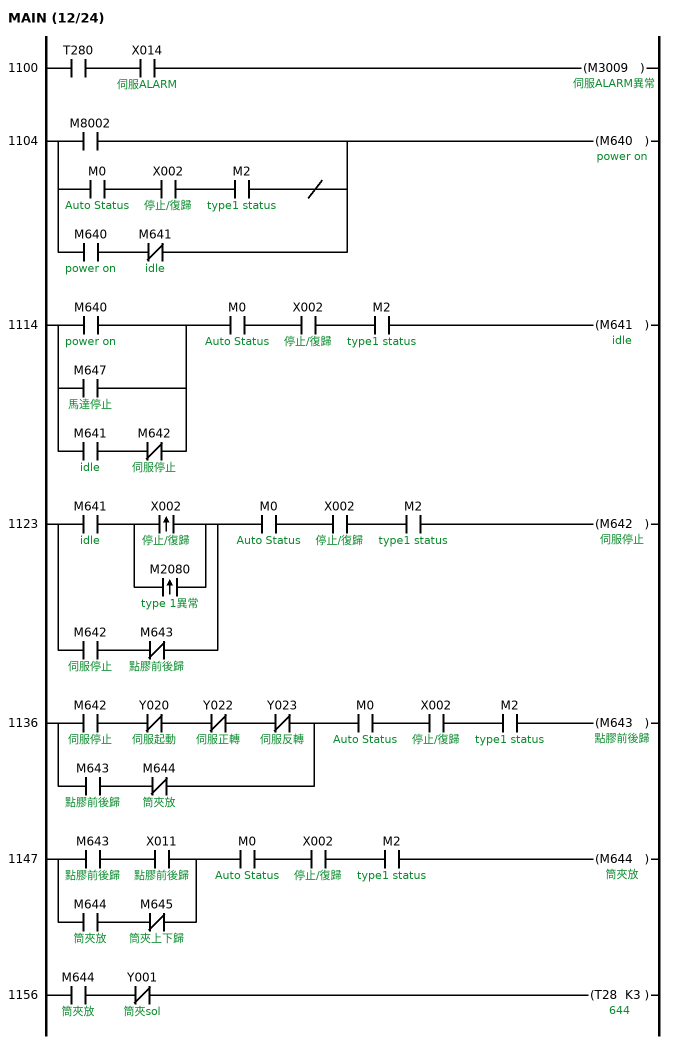
1100  LD      T280
      AND     X014  ; 伺服ALARM
      OUT     M3009  ; 伺服ALARM異常
1104  LD      M8002
      LD      M0  ; Auto Status
      AND     X002  ; 停止/復歸
      AND     M2  ; type1 status
      INV
      ORB
      LD      M640  ; power on
      ANI     M641  ; idle
      ORB
      OUT     M640  ; power on
1114  LD      M640  ; power on
      OR      M647  ; 馬達停止
      LD      M641  ; idle
      ANI     M642  ; 伺服停止
      ORB
      AND     M0  ; Auto Status
      AND     X002  ; 停止/復歸
      AND     M2  ; type1 status
      OUT     M641  ; idle
1123  LD      M641  ; idle
      LDP     X002  ; 停止/復歸
      ORP     M2080  ; type 1異常
      ANB
      LD      M642  ; 伺服停止
      ANI     M643  ; 點膠前後歸
      ORB
      AND     M0  ; Auto Status
      AND     X002  ; 停止/復歸
      AND     M2  ; type1 status
      OUT     M642  ; 伺服停止
1136  LD      M642  ; 伺服停止
      ANI     Y020  ; 伺服起動
      ANI     Y022  ; 伺服正轉
      ANI     Y023  ; 伺服反轉
      LD      M643  ; 點膠前後歸
      ANI     M644  ; 筒夾放
      ORB
      AND     M0  ; Auto Status
      AND     X002  ; 停止/復歸
      AND     M2  ; type1 status
      OUT     M643  ; 點膠前後歸
1147  LD      M643  ; 點膠前後歸
      AND     X011  ; 點膠前後歸
      LD      M644  ; 筒夾放
      ANI     M645  ; 筒夾上下歸
      ORB
      AND     M0  ; Auto Status
      AND     X002  ; 停止/復歸
      AND     M2  ; type1 status
      OUT     M644  ; 筒夾放
1156  LD      M644  ; 筒夾放
      ANI     Y001  ; 筒夾sol
      OUT     T28 K3  ; 644
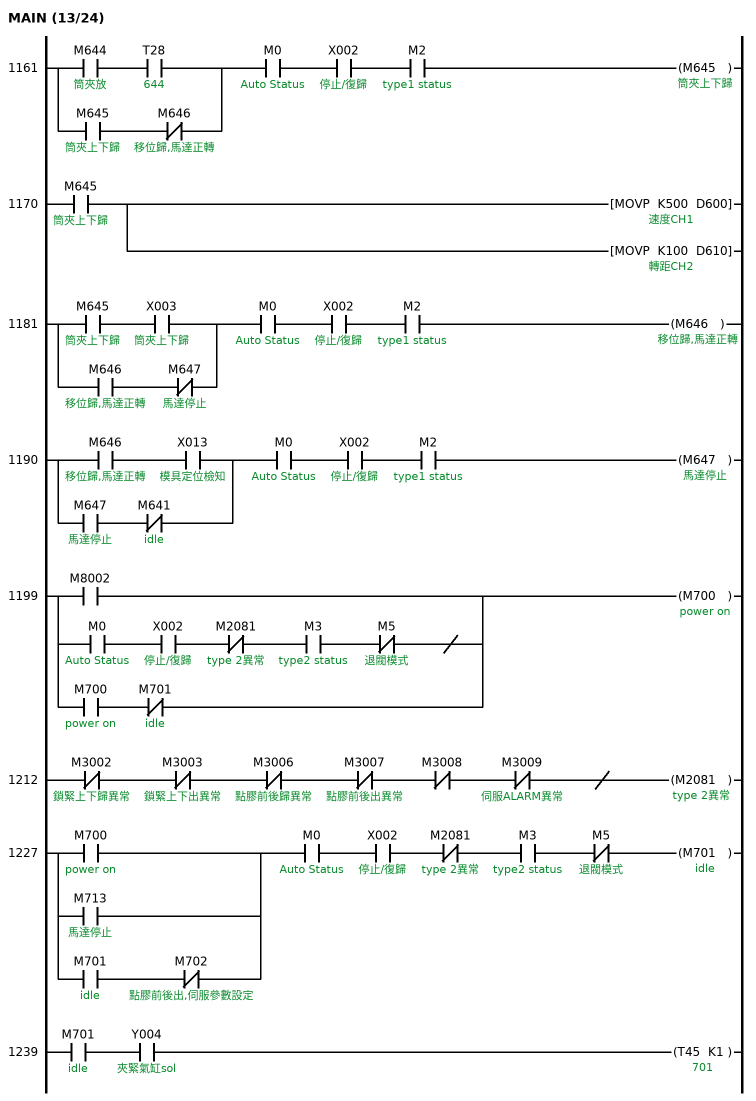
1161  LD      M644  ; 筒夾放
      AND     T28  ; 644
      LD      M645  ; 筒夾上下歸
      ANI     M646  ; 移位歸,馬達正轉
      ORB
      AND     M0  ; Auto Status
      AND     X002  ; 停止/復歸
      AND     M2  ; type1 status
      OUT     M645  ; 筒夾上下歸
1170  LD      M645  ; 筒夾上下歸
      MOVP    K500 D600
      MOVP    K100 D610
1181  LD      M645  ; 筒夾上下歸
      AND     X003  ; 筒夾上下歸
      LD      M646  ; 移位歸,馬達正轉
      ANI     M647  ; 馬達停止
      ORB
      AND     M0  ; Auto Status
      AND     X002  ; 停止/復歸
      AND     M2  ; type1 status
      OUT     M646  ; 移位歸,馬達正轉
1190  LD      M646  ; 移位歸,馬達正轉
      AND     X013  ; 模具定位檢知
      LD      M647  ; 馬達停止
      ANI     M641  ; idle
      ORB
      AND     M0  ; Auto Status
      AND     X002  ; 停止/復歸
      AND     M2  ; type1 status
      OUT     M647  ; 馬達停止
1199  LD      M8002
      LD      M0  ; Auto Status
      AND     X002  ; 停止/復歸
      ANI     M2081  ; type 2異常
      AND     M3  ; type2 status
      ANI     M5  ; 退閥模式
      INV
      ORB
      LD      M700  ; power on
      ANI     M701  ; idle
      ORB
      OUT     M700  ; power on
1212  LDI     M3002  ; 鎖緊上下歸異常
      ANI     M3003  ; 鎖緊上下出異常
      ANI     M3006  ; 點膠前後歸異常
      ANI     M3007  ; 點膠前後出異常
      ANI     M3008
      ANI     M3009  ; 伺服ALARM異常
      INV
      OUT     M2081  ; type 2異常
1227  LD      M700  ; power on
      OR      M713  ; 馬達停止
      LD      M701  ; idle
      ANI     M702  ; 點膠前後出,伺服參數設定
      ORB
      AND     M0  ; Auto Status
      AND     X002  ; 停止/復歸
      ANI     M2081  ; type 2異常
      AND     M3  ; type2 status
      ANI     M5  ; 退閥模式
      OUT     M701  ; idle
1239  LD      M701  ; idle
      AND     Y004  ; 夾緊氣缸sol
      OUT     T45 K1  ; 701
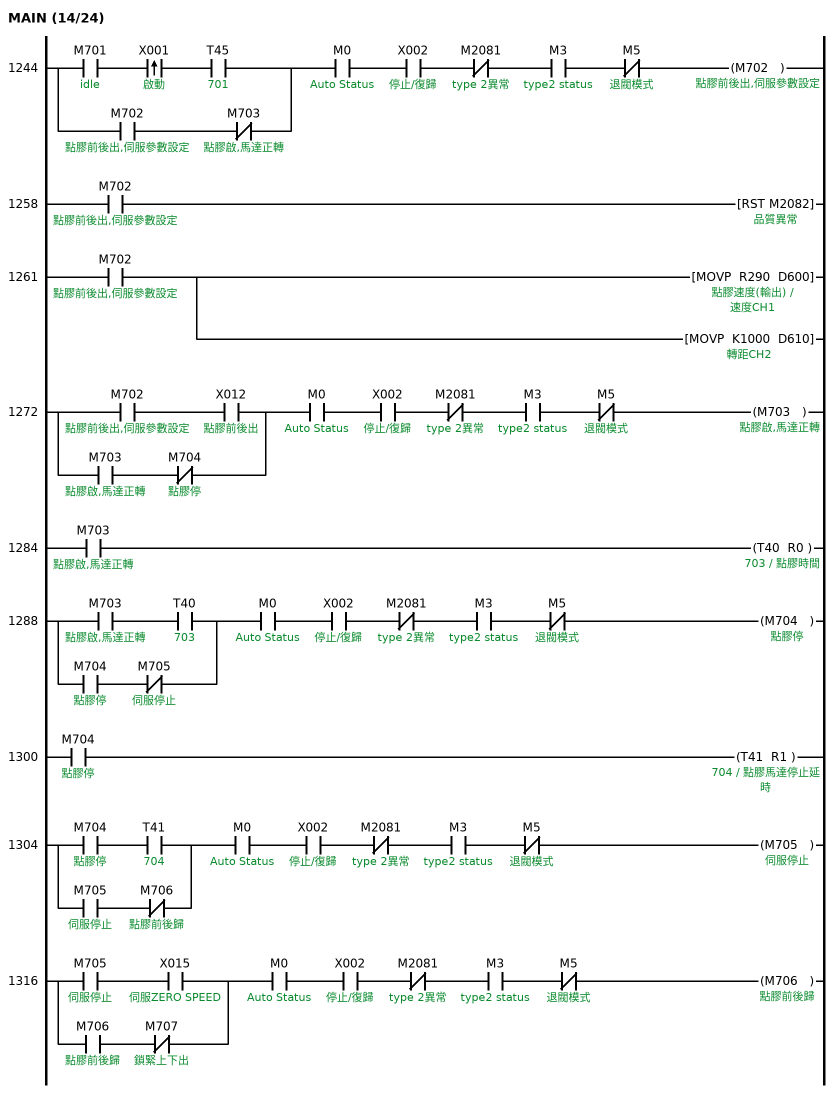
1244  LD      M701  ; idle
      ANDP    X001  ; 啟動
      AND     T45  ; 701
      LD      M702  ; 點膠前後出,伺服參數設定
      ANI     M703  ; 點膠啟,馬達正轉
      ORB
      AND     M0  ; Auto Status
      AND     X002  ; 停止/復歸
      ANI     M2081  ; type 2異常
      AND     M3  ; type2 status
      ANI     M5  ; 退閥模式
      OUT     M702  ; 點膠前後出,伺服參數設定
1258  LD      M702  ; 點膠前後出,伺服參數設定
      RST     M2082  ; 品質異常
1261  LD      M702  ; 點膠前後出,伺服參數設定
      MOVP    R290 D600
      MOVP    K1000 D610
1272  LD      M702  ; 點膠前後出,伺服參數設定
      AND     X012  ; 點膠前後出
      LD      M703  ; 點膠啟,馬達正轉
      ANI     M704  ; 點膠停
      ORB
      AND     M0  ; Auto Status
      AND     X002  ; 停止/復歸
      ANI     M2081  ; type 2異常
      AND     M3  ; type2 status
      ANI     M5  ; 退閥模式
      OUT     M703  ; 點膠啟,馬達正轉
1284  LD      M703  ; 點膠啟,馬達正轉
      OUT     T40 R0  ; 703 / 點膠時間
1288  LD      M703  ; 點膠啟,馬達正轉
      AND     T40  ; 703
      LD      M704  ; 點膠停
      ANI     M705  ; 伺服停止
      ORB
      AND     M0  ; Auto Status
      AND     X002  ; 停止/復歸
      ANI     M2081  ; type 2異常
      AND     M3  ; type2 status
      ANI     M5  ; 退閥模式
      OUT     M704  ; 點膠停
1300  LD      M704  ; 點膠停
      OUT     T41 R1  ; 704 / 點膠馬達停止延時
1304  LD      M704  ; 點膠停
      AND     T41  ; 704
      LD      M705  ; 伺服停止
      ANI     M706  ; 點膠前後歸
      ORB
      AND     M0  ; Auto Status
      AND     X002  ; 停止/復歸
      ANI     M2081  ; type 2異常
      AND     M3  ; type2 status
      ANI     M5  ; 退閥模式
      OUT     M705  ; 伺服停止
1316  LD      M705  ; 伺服停止
      AND     X015  ; 伺服ZERO SPEED
      LD      M706  ; 點膠前後歸
      ANI     M707  ; 鎖緊上下出
      ORB
      AND     M0  ; Auto Status
      AND     X002  ; 停止/復歸
      ANI     M2081  ; type 2異常
      AND     M3  ; type2 status
      ANI     M5  ; 退閥模式
      OUT     M706  ; 點膠前後歸
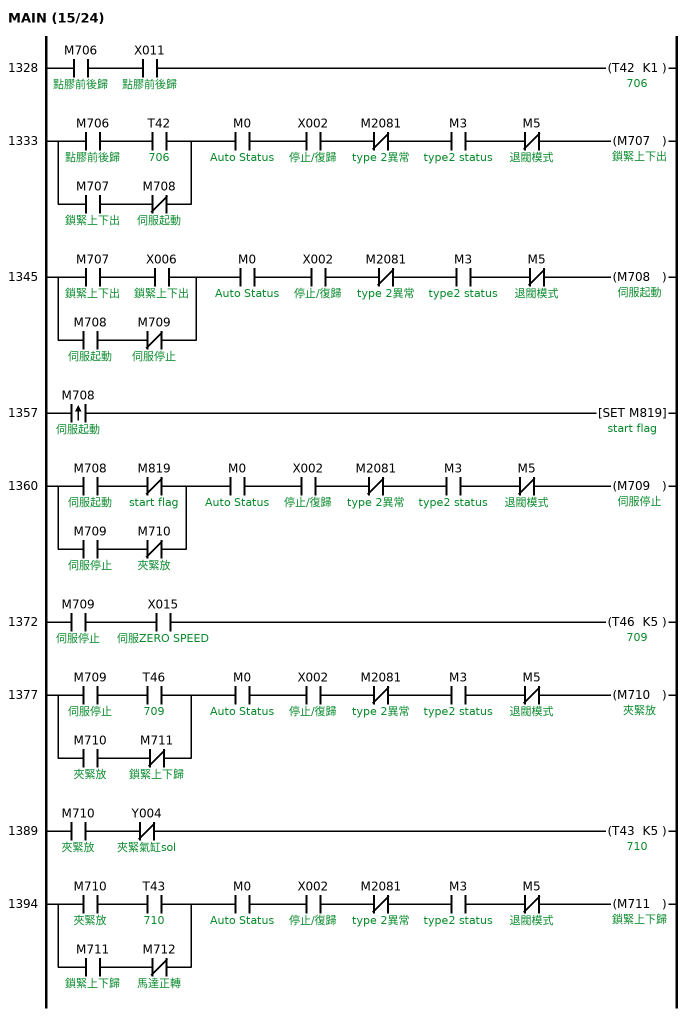
1328  LD      M706  ; 點膠前後歸
      AND     X011  ; 點膠前後歸
      OUT     T42 K1  ; 706
1333  LD      M706  ; 點膠前後歸
      AND     T42  ; 706
      LD      M707  ; 鎖緊上下出
      ANI     M708  ; 伺服起動
      ORB
      AND     M0  ; Auto Status
      AND     X002  ; 停止/復歸
      ANI     M2081  ; type 2異常
      AND     M3  ; type2 status
      ANI     M5  ; 退閥模式
      OUT     M707  ; 鎖緊上下出
1345  LD      M707  ; 鎖緊上下出
      AND     X006  ; 鎖緊上下出
      LD      M708  ; 伺服起動
      ANI     M709  ; 伺服停止
      ORB
      AND     M0  ; Auto Status
      AND     X002  ; 停止/復歸
      ANI     M2081  ; type 2異常
      AND     M3  ; type2 status
      ANI     M5  ; 退閥模式
      OUT     M708  ; 伺服起動
1357  LDP     M708  ; 伺服起動
      SET     M819  ; start flag
1360  LD      M708  ; 伺服起動
      ANI     M819  ; start flag
      LD      M709  ; 伺服停止
      ANI     M710  ; 夾緊放
      ORB
      AND     M0  ; Auto Status
      AND     X002  ; 停止/復歸
      ANI     M2081  ; type 2異常
      AND     M3  ; type2 status
      ANI     M5  ; 退閥模式
      OUT     M709  ; 伺服停止
1372  LD      M709  ; 伺服停止
      AND     X015  ; 伺服ZERO SPEED
      OUT     T46 K5  ; 709
1377  LD      M709  ; 伺服停止
      AND     T46  ; 709
      LD      M710  ; 夾緊放
      ANI     M711  ; 鎖緊上下歸
      ORB
      AND     M0  ; Auto Status
      AND     X002  ; 停止/復歸
      ANI     M2081  ; type 2異常
      AND     M3  ; type2 status
      ANI     M5  ; 退閥模式
      OUT     M710  ; 夾緊放
1389  LD      M710  ; 夾緊放
      ANI     Y004  ; 夾緊氣缸sol
      OUT     T43 K5  ; 710
1394  LD      M710  ; 夾緊放
      AND     T43  ; 710
      LD      M711  ; 鎖緊上下歸
      ANI     M712  ; 馬達正轉
      ORB
      AND     M0  ; Auto Status
      AND     X002  ; 停止/復歸
      ANI     M2081  ; type 2異常
      AND     M3  ; type2 status
      ANI     M5  ; 退閥模式
      OUT     M711  ; 鎖緊上下歸
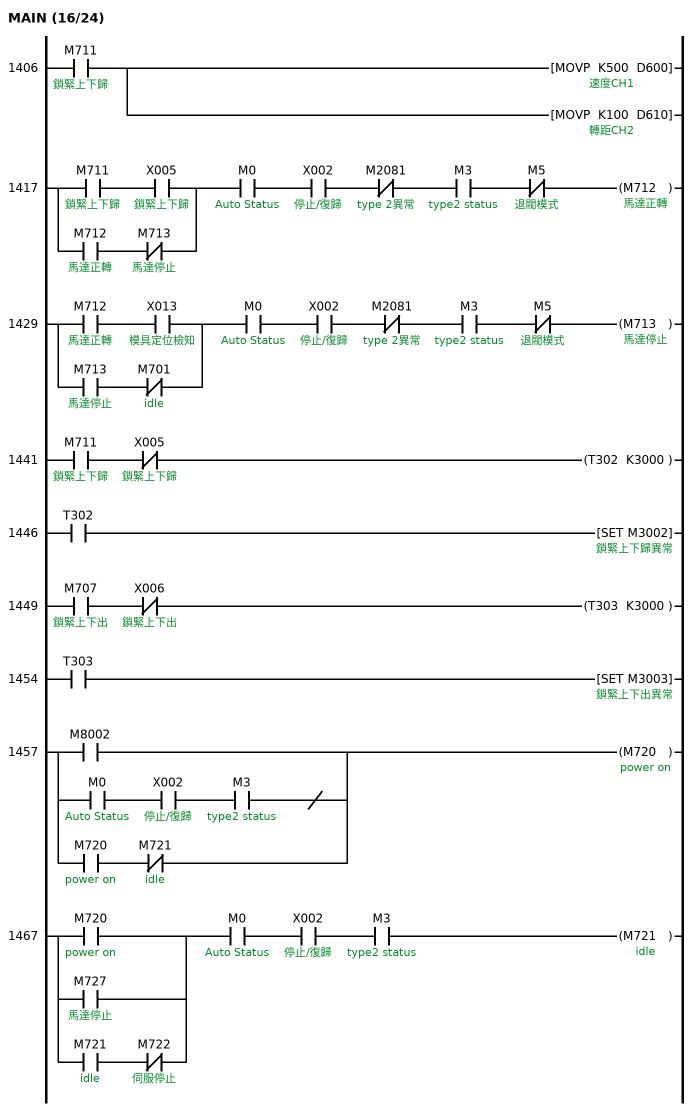
1406  LD      M711  ; 鎖緊上下歸
      MOVP    K500 D600
      MOVP    K100 D610
1417  LD      M711  ; 鎖緊上下歸
      AND     X005  ; 鎖緊上下歸
      LD      M712  ; 馬達正轉
      ANI     M713  ; 馬達停止
      ORB
      AND     M0  ; Auto Status
      AND     X002  ; 停止/復歸
      ANI     M2081  ; type 2異常
      AND     M3  ; type2 status
      ANI     M5  ; 退閥模式
      OUT     M712  ; 馬達正轉
1429  LD      M712  ; 馬達正轉
      AND     X013  ; 模具定位檢知
      LD      M713  ; 馬達停止
      ANI     M701  ; idle
      ORB
      AND     M0  ; Auto Status
      AND     X002  ; 停止/復歸
      ANI     M2081  ; type 2異常
      AND     M3  ; type2 status
      ANI     M5  ; 退閥模式
      OUT     M713  ; 馬達停止
1441  LD      M711  ; 鎖緊上下歸
      ANI     X005  ; 鎖緊上下歸
      OUT     T302 K3000
1446  LD      T302
      SET     M3002  ; 鎖緊上下歸異常
1449  LD      M707  ; 鎖緊上下出
      ANI     X006  ; 鎖緊上下出
      OUT     T303 K3000
1454  LD      T303
      SET     M3003  ; 鎖緊上下出異常
1457  LD      M8002
      LD      M0  ; Auto Status
      AND     X002  ; 停止/復歸
      AND     M3  ; type2 status
      INV
      ORB
      LD      M720  ; power on
      ANI     M721  ; idle
      ORB
      OUT     M720  ; power on
1467  LD      M720  ; power on
      OR      M727  ; 馬達停止
      LD      M721  ; idle
      ANI     M722  ; 伺服停止
      ORB
      AND     M0  ; Auto Status
      AND     X002  ; 停止/復歸
      AND     M3  ; type2 status
      OUT     M721  ; idle
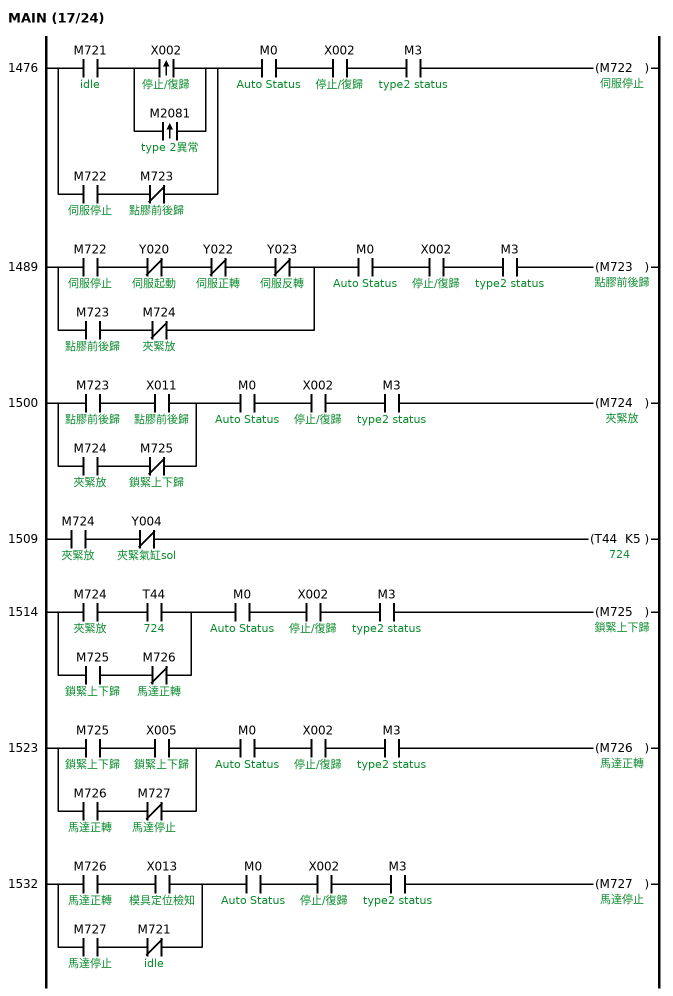
1476  LD      M721  ; idle
      LDP     X002  ; 停止/復歸
      ORP     M2081  ; type 2異常
      ANB
      LD      M722  ; 伺服停止
      ANI     M723  ; 點膠前後歸
      ORB
      AND     M0  ; Auto Status
      AND     X002  ; 停止/復歸
      AND     M3  ; type2 status
      OUT     M722  ; 伺服停止
1489  LD      M722  ; 伺服停止
      ANI     Y020  ; 伺服起動
      ANI     Y022  ; 伺服正轉
      ANI     Y023  ; 伺服反轉
      LD      M723  ; 點膠前後歸
      ANI     M724  ; 夾緊放
      ORB
      AND     M0  ; Auto Status
      AND     X002  ; 停止/復歸
      AND     M3  ; type2 status
      OUT     M723  ; 點膠前後歸
1500  LD      M723  ; 點膠前後歸
      AND     X011  ; 點膠前後歸
      LD      M724  ; 夾緊放
      ANI     M725  ; 鎖緊上下歸
      ORB
      AND     M0  ; Auto Status
      AND     X002  ; 停止/復歸
      AND     M3  ; type2 status
      OUT     M724  ; 夾緊放
1509  LD      M724  ; 夾緊放
      ANI     Y004  ; 夾緊氣缸sol
      OUT     T44 K5  ; 724
1514  LD      M724  ; 夾緊放
      AND     T44  ; 724
      LD      M725  ; 鎖緊上下歸
      ANI     M726  ; 馬達正轉
      ORB
      AND     M0  ; Auto Status
      AND     X002  ; 停止/復歸
      AND     M3  ; type2 status
      OUT     M725  ; 鎖緊上下歸
1523  LD      M725  ; 鎖緊上下歸
      AND     X005  ; 鎖緊上下歸
      LD      M726  ; 馬達正轉
      ANI     M727  ; 馬達停止
      ORB
      AND     M0  ; Auto Status
      AND     X002  ; 停止/復歸
      AND     M3  ; type2 status
      OUT     M726  ; 馬達正轉
1532  LD      M726  ; 馬達正轉
      AND     X013  ; 模具定位檢知
      LD      M727  ; 馬達停止
      ANI     M721  ; idle
      ORB
      AND     M0  ; Auto Status
      AND     X002  ; 停止/復歸
      AND     M3  ; type2 status
      OUT     M727  ; 馬達停止
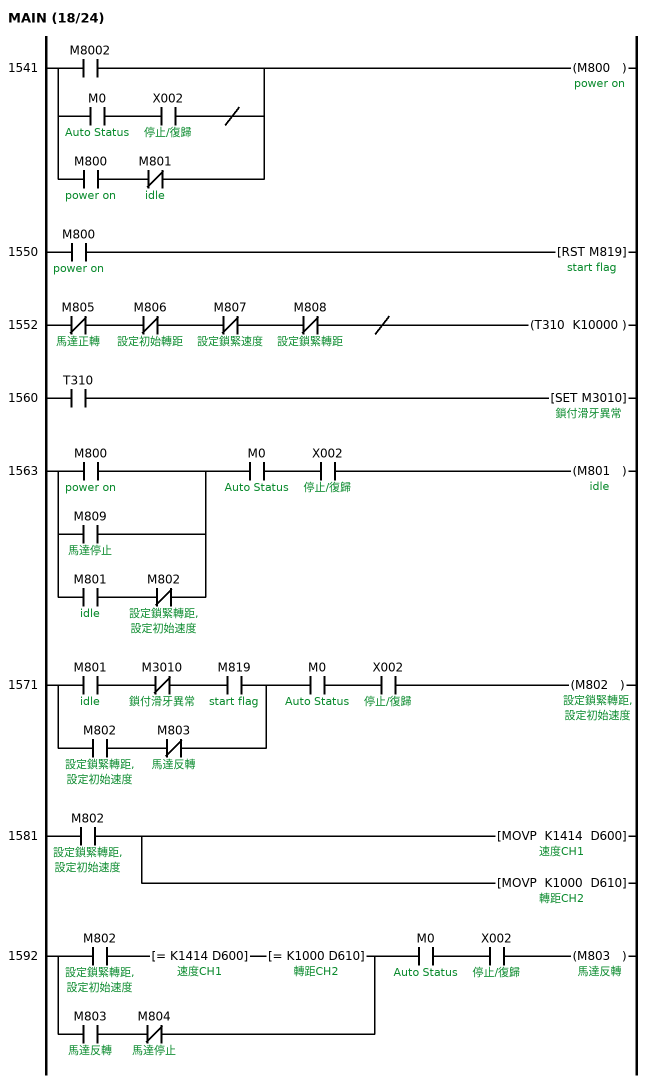
1541  LD      M8002
      LD      M0  ; Auto Status
      AND     X002  ; 停止/復歸
      INV
      ORB
      LD      M800  ; power on
      ANI     M801  ; idle
      ORB
      OUT     M800  ; power on
1550  LD      M800  ; power on
      RST     M819  ; start flag
1552  LDI     M805  ; 馬達正轉
      ANI     M806  ; 設定初始轉距
      ANI     M807  ; 設定鎖緊速度
      ANI     M808  ; 設定鎖緊轉距
      INV
      OUT     T310 K10000
1560  LD      T310
      SET     M3010  ; 鎖付滑牙異常
1563  LD      M800  ; power on
      OR      M809  ; 馬達停止
      LD      M801  ; idle
      ANI     M802  ; 設定鎖緊轉距,設定初始速度
      ORB
      AND     M0  ; Auto Status
      AND     X002  ; 停止/復歸
      OUT     M801  ; idle
1571  LD      M801  ; idle
      ANI     M3010  ; 鎖付滑牙異常
      AND     M819  ; start flag
      LD      M802  ; 設定鎖緊轉距,設定初始速度
      ANI     M803  ; 馬達反轉
      ORB
      AND     M0  ; Auto Status
      AND     X002  ; 停止/復歸
      OUT     M802  ; 設定鎖緊轉距,設定初始速度
1581  LD      M802  ; 設定鎖緊轉距,設定初始速度
      MOVP    K1414 D600
      MOVP    K1000 D610
1592  LD      M802  ; 設定鎖緊轉距,設定初始速度
      AND=    K1414 D600  ; 速度CH1
      AND=    K1000 D610  ; 轉距CH2
      LD      M803  ; 馬達反轉
      ANI     M804  ; 馬達停止
      ORB
      AND     M0  ; Auto Status
      AND     X002  ; 停止/復歸
      OUT     M803  ; 馬達反轉
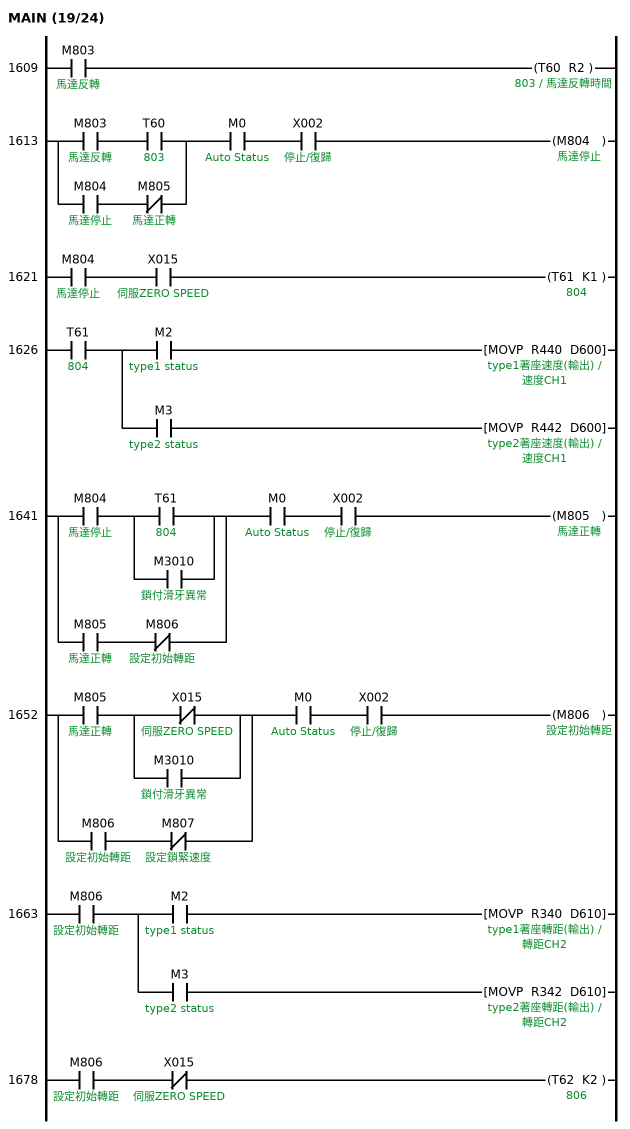
1609  LD      M803  ; 馬達反轉
      OUT     T60 R2  ; 803 / 馬達反轉時間
1613  LD      M803  ; 馬達反轉
      AND     T60  ; 803
      LD      M804  ; 馬達停止
      ANI     M805  ; 馬達正轉
      ORB
      AND     M0  ; Auto Status
      AND     X002  ; 停止/復歸
      OUT     M804  ; 馬達停止
1621  LD      M804  ; 馬達停止
      AND     X015  ; 伺服ZERO SPEED
      OUT     T61 K1  ; 804
1626  LD      T61  ; 804
      MPS
      AND     M2  ; type1 status
      MOVP    R440 D600  ; type1著座速度(輸出)
      MPP
      AND     M3  ; type2 status
      MOVP    R442 D600  ; type2著座速度(輸出)
1641  LD      M804  ; 馬達停止
      LD      T61  ; 804
      OR      M3010  ; 鎖付滑牙異常
      ANB
      LD      M805  ; 馬達正轉
      ANI     M806  ; 設定初始轉距
      ORB
      AND     M0  ; Auto Status
      AND     X002  ; 停止/復歸
      OUT     M805  ; 馬達正轉
1652  LD      M805  ; 馬達正轉
      LDI     X015  ; 伺服ZERO SPEED
      OR      M3010  ; 鎖付滑牙異常
      ANB
      LD      M806  ; 設定初始轉距
      ANI     M807  ; 設定鎖緊速度
      ORB
      AND     M0  ; Auto Status
      AND     X002  ; 停止/復歸
      OUT     M806  ; 設定初始轉距
1663  LD      M806  ; 設定初始轉距
      MPS
      AND     M2  ; type1 status
      MOVP    R340 D610  ; type1著座轉距(輸出)
      MPP
      AND     M3  ; type2 status
      MOVP    R342 D610  ; type2著座轉距(輸出)
1678  LD      M806  ; 設定初始轉距
      ANI     X015  ; 伺服ZERO SPEED
      OUT     T62 K2  ; 806
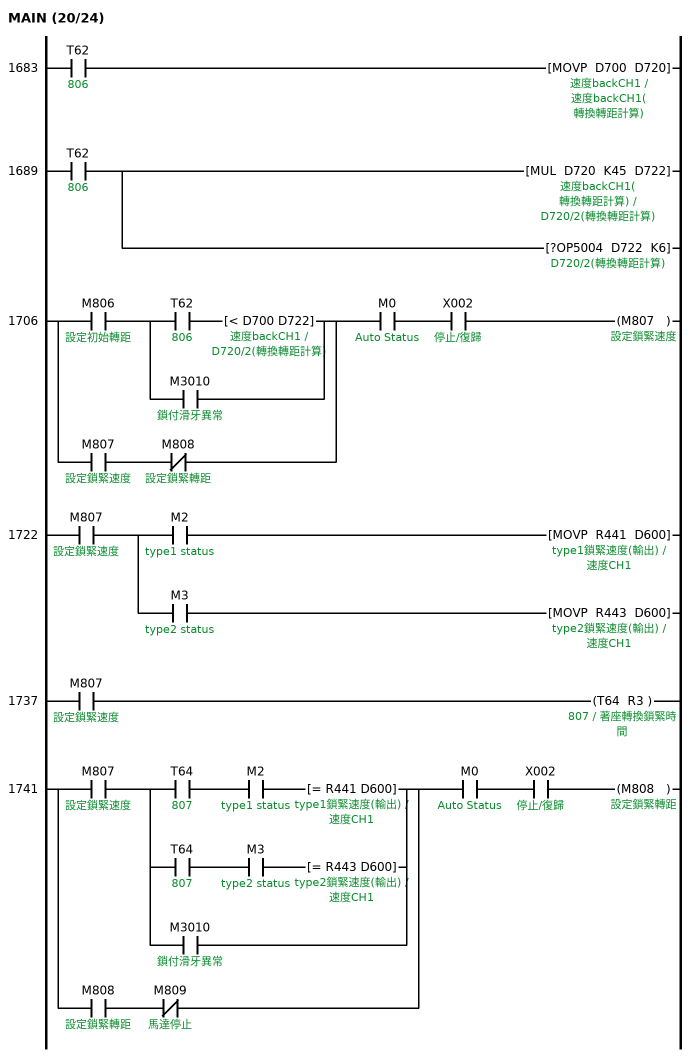
1683  LD      T62  ; 806
      MOVP    D700 D720  ; 速度backCH1(轉換轉距計算)
1689  LD      T62  ; 806
      MUL     D720 K45 D722  ; D720/2(轉換轉距計算)
      ?OP5004 D722 K6
1706  LD      M806  ; 設定初始轉距
      LD      T62  ; 806
      AND<    D700 D722  ; 速度backCH1 / D720/2(轉換轉距計算)
      OR      M3010  ; 鎖付滑牙異常
      ANB
      LD      M807  ; 設定鎖緊速度
      ANI     M808  ; 設定鎖緊轉距
      ORB
      AND     M0  ; Auto Status
      AND     X002  ; 停止/復歸
      OUT     M807  ; 設定鎖緊速度
1722  LD      M807  ; 設定鎖緊速度
      MPS
      AND     M2  ; type1 status
      MOVP    R441 D600  ; type1鎖緊速度(輸出)
      MPP
      AND     M3  ; type2 status
      MOVP    R443 D600  ; type2鎖緊速度(輸出)
1737  LD      M807  ; 設定鎖緊速度
      OUT     T64 R3  ; 807 / 著座轉換鎖緊時間
1741  LD      M807  ; 設定鎖緊速度
      LD      T64  ; 807
      AND     M2  ; type1 status
      AND=    R441 D600  ; type1鎖緊速度(輸出) / 速度CH1
      LD      T64  ; 807
      AND     M3  ; type2 status
      AND=    R443 D600  ; type2鎖緊速度(輸出) / 速度CH1
      ORB
      OR      M3010  ; 鎖付滑牙異常
      ANB
      LD      M808  ; 設定鎖緊轉距
      ANI     M809  ; 馬達停止
      ORB
      AND     M0  ; Auto Status
      AND     X002  ; 停止/復歸
      OUT     M808  ; 設定鎖緊轉距
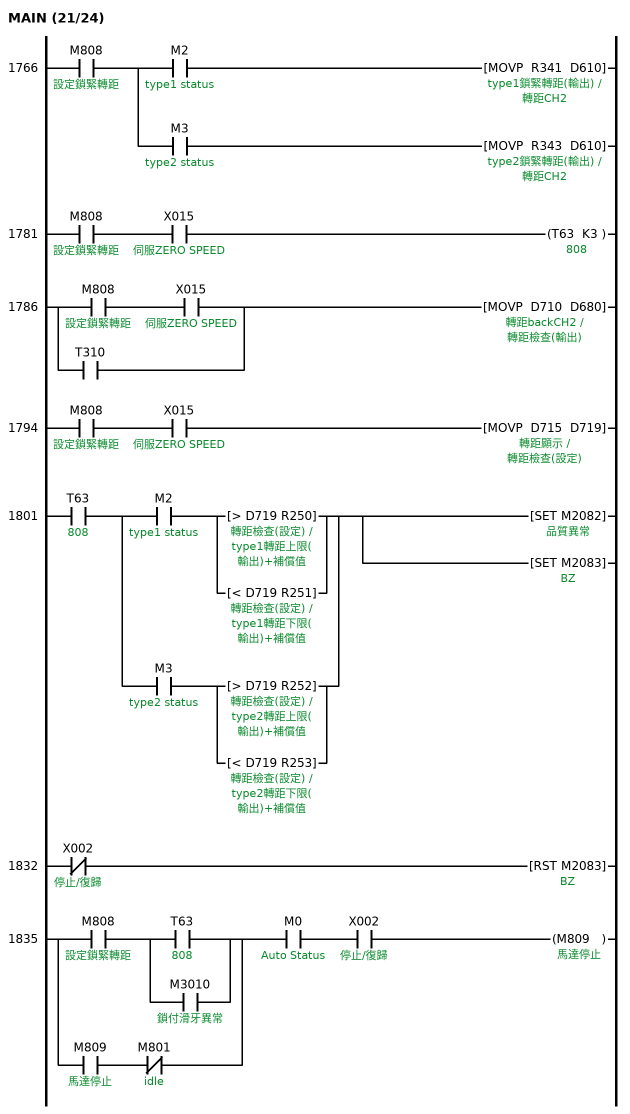
1766  LD      M808  ; 設定鎖緊轉距
      MPS
      AND     M2  ; type1 status
      MOVP    R341 D610  ; type1鎖緊轉距(輸出)
      MPP
      AND     M3  ; type2 status
      MOVP    R343 D610  ; type2鎖緊轉距(輸出)
1781  LD      M808  ; 設定鎖緊轉距
      AND     X015  ; 伺服ZERO SPEED
      OUT     T63 K3  ; 808
1786  LD      M808  ; 設定鎖緊轉距
      AND     X015  ; 伺服ZERO SPEED
      OR      T310
      MOVP    D710 D680  ; 轉距檢查(輸出)
1794  LD      M808  ; 設定鎖緊轉距
      AND     X015  ; 伺服ZERO SPEED
      MOVP    D715 D719  ; 轉距顯示 / 轉距檢查(設定)
1801  LD      T63  ; 808
      LD      M2  ; type1 status
      LD>     D719 R250  ; 轉距檢查(設定) / type1轉距上限(輸出)+補償值
      OR<     D719 R251  ; 轉距檢查(設定) / type1轉距下限(輸出)+補償值
      ANB
      LD      M3  ; type2 status
      LD>     D719 R252  ; 轉距檢查(設定) / type2轉距上限(輸出)+補償值
      OR<     D719 R253  ; 轉距檢查(設定) / type2轉距下限(輸出)+補償值
      ANB
      ORB
      ANB
      SET     M2082  ; 品質異常
      SET     M2083  ; BZ
1832  LDI     X002  ; 停止/復歸
      RST     M2083  ; BZ
1835  LD      M808  ; 設定鎖緊轉距
      LD      T63  ; 808
      OR      M3010  ; 鎖付滑牙異常
      ANB
      LD      M809  ; 馬達停止
      ANI     M801  ; idle
      ORB
      AND     M0  ; Auto Status
      AND     X002  ; 停止/復歸
      OUT     M809  ; 馬達停止
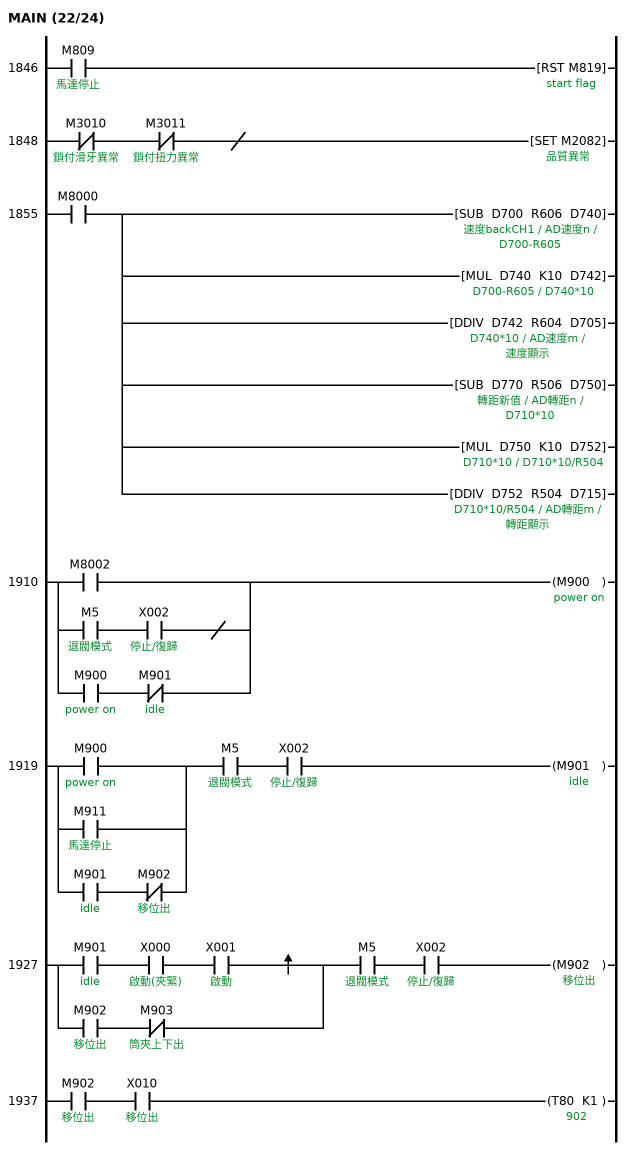
1846  LD      M809  ; 馬達停止
      RST     M819  ; start flag
1848  LDI     M3010  ; 鎖付滑牙異常
      ANI     M3011  ; 鎖付扭力異常
      INV
      SET     M2082  ; 品質異常
1855  LD      M8000
      SUB     D700 R606 D740  ; AD速度n / D700-R605
      MUL     D740 K10 D742  ; D740*10
      DDIV    D742 R604 D705  ; AD速度m / 速度顯示
      SUB     D770 R506 D750  ; AD轉距n / D710*10
      MUL     D750 K10 D752  ; D710*10/R504
      DDIV    D752 R504 D715  ; AD轉距m
1910  LD      M8002
      LD      M5  ; 退閥模式
      AND     X002  ; 停止/復歸
      INV
      ORB
      LD      M900  ; power on
      ANI     M901  ; idle
      ORB
      OUT     M900  ; power on
1919  LD      M900  ; power on
      OR      M911  ; 馬達停止
      LD      M901  ; idle
      ANI     M902  ; 移位出
      ORB
      AND     M5  ; 退閥模式
      AND     X002  ; 停止/復歸
      OUT     M901  ; idle
1927  LD      M901  ; idle
      AND     X000  ; 啟動(夾緊)
      AND     X001  ; 啟動
      MEP
      LD      M902  ; 移位出
      ANI     M903  ; 筒夾上下出
      ORB
      AND     M5  ; 退閥模式
      AND     X002  ; 停止/復歸
      OUT     M902  ; 移位出
1937  LD      M902  ; 移位出
      AND     X010  ; 移位出
      OUT     T80 K1  ; 902
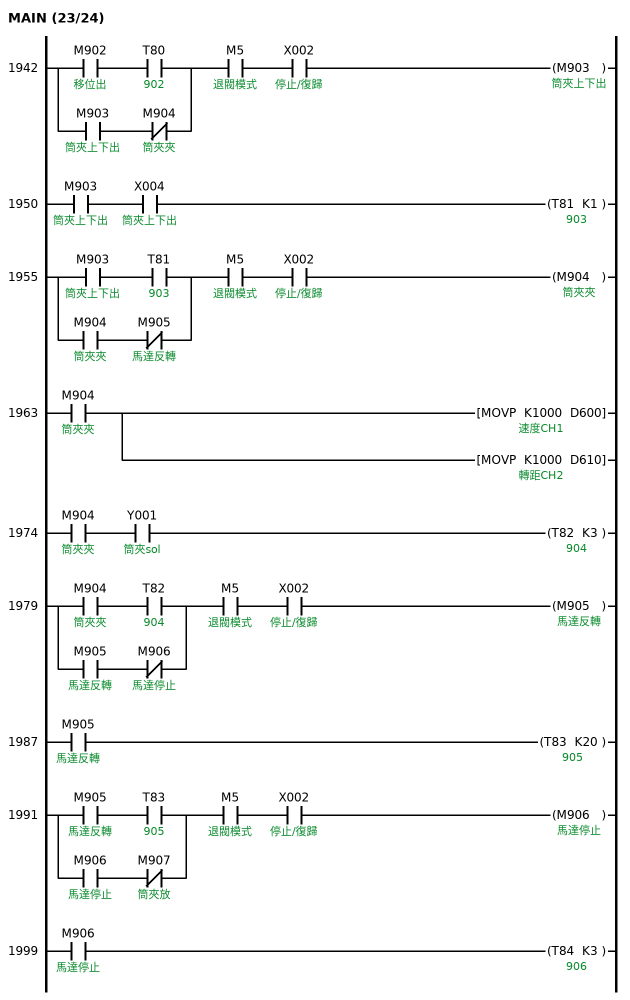
1942  LD      M902  ; 移位出
      AND     T80  ; 902
      LD      M903  ; 筒夾上下出
      ANI     M904  ; 筒夾夾
      ORB
      AND     M5  ; 退閥模式
      AND     X002  ; 停止/復歸
      OUT     M903  ; 筒夾上下出
1950  LD      M903  ; 筒夾上下出
      AND     X004  ; 筒夾上下出
      OUT     T81 K1  ; 903
1955  LD      M903  ; 筒夾上下出
      AND     T81  ; 903
      LD      M904  ; 筒夾夾
      ANI     M905  ; 馬達反轉
      ORB
      AND     M5  ; 退閥模式
      AND     X002  ; 停止/復歸
      OUT     M904  ; 筒夾夾
1963  LD      M904  ; 筒夾夾
      MOVP    K1000 D600
      MOVP    K1000 D610
1974  LD      M904  ; 筒夾夾
      AND     Y001  ; 筒夾sol
      OUT     T82 K3  ; 904
1979  LD      M904  ; 筒夾夾
      AND     T82  ; 904
      LD      M905  ; 馬達反轉
      ANI     M906  ; 馬達停止
      ORB
      AND     M5  ; 退閥模式
      AND     X002  ; 停止/復歸
      OUT     M905  ; 馬達反轉
1987  LD      M905  ; 馬達反轉
      OUT     T83 K20  ; 905
1991  LD      M905  ; 馬達反轉
      AND     T83  ; 905
      LD      M906  ; 馬達停止
      ANI     M907  ; 筒夾放
      ORB
      AND     M5  ; 退閥模式
      AND     X002  ; 停止/復歸
      OUT     M906  ; 馬達停止
1999  LD      M906  ; 馬達停止
      OUT     T84 K3  ; 906
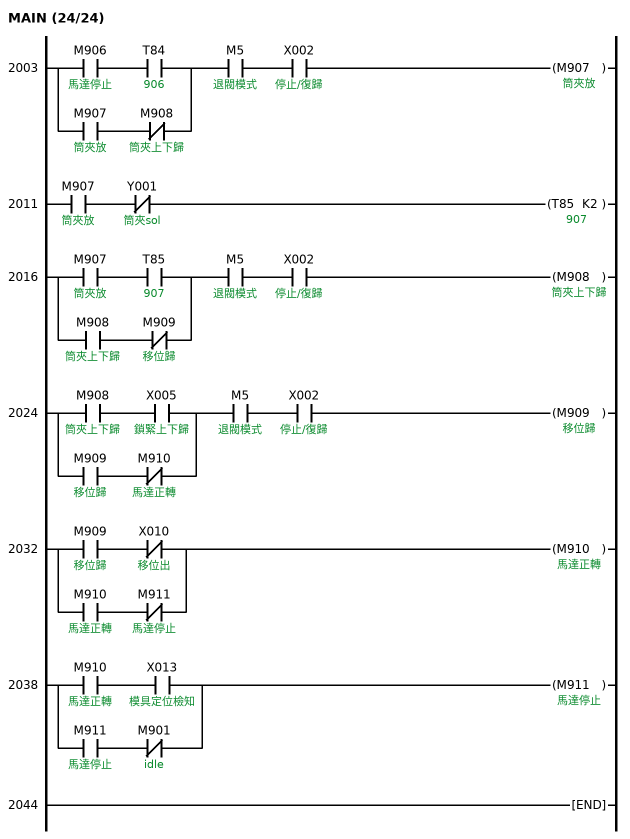
2003  LD      M906  ; 馬達停止
      AND     T84  ; 906
      LD      M907  ; 筒夾放
      ANI     M908  ; 筒夾上下歸
      ORB
      AND     M5  ; 退閥模式
      AND     X002  ; 停止/復歸
      OUT     M907  ; 筒夾放
2011  LD      M907  ; 筒夾放
      ANI     Y001  ; 筒夾sol
      OUT     T85 K2  ; 907
2016  LD      M907  ; 筒夾放
      AND     T85  ; 907
      LD      M908  ; 筒夾上下歸
      ANI     M909  ; 移位歸
      ORB
      AND     M5  ; 退閥模式
      AND     X002  ; 停止/復歸
      OUT     M908  ; 筒夾上下歸
2024  LD      M908  ; 筒夾上下歸
      AND     X005  ; 鎖緊上下歸
      LD      M909  ; 移位歸
      ANI     M910  ; 馬達正轉
      ORB
      AND     M5  ; 退閥模式
      AND     X002  ; 停止/復歸
      OUT     M909  ; 移位歸
2032  LD      M909  ; 移位歸
      ANI     X010  ; 移位出
      LD      M910  ; 馬達正轉
      ANI     M911  ; 馬達停止
      ORB
      OUT     M910  ; 馬達正轉
2038  LD      M910  ; 馬達正轉
      AND     X013  ; 模具定位檢知
      LD      M911  ; 馬達停止
      ANI     M901  ; idle
      ORB
      OUT     M911  ; 馬達停止
2044  END
END_PROGRAM

// device comments not shown above
M6  ; 退閥啟動
M502  ; 筒夾放鬆PB
M505  ; 夾緊氣缸放PB
M511  ; 伺服異常重置PB
D723  ; **************
D778  ; D776/10
R201  ; ******
R240  ; type1轉距補償(輸出)
R241  ; type2轉距補償(輸出)
R260  ; 手動速度(設定)
R261  ; 手動轉距(設定)
R270  ; 點膠速度(設定)
R304  ; DA轉距m
R305  ; DA轉距n
R380  ; type1轉距上限(輸出)
R381  ; type1轉距下限(輸出)
R382  ; type2轉距上限(輸出)
R383  ; type2轉距下限(輸出)
R404  ; DA速度m
R405  ; DA速度n
R1000  ; #1著座速度(set)
R1002  ; #1鎖緊速度(set)
R1004  ; #1著座扭力(set)
R1006  ; #1鎖緊扭力(set)
R1008  ; #1扭力上限(set)
R1010  ; #1扭力下限(set)
R1012  ; #1扭力補償(set)
R1020  ; #1著座速度(output)
R1022  ; #1鎖緊速度(output)
R1024  ; #1著座扭力(output)
R1026  ; #1鎖緊扭力(output)
R1028  ; #1扭力上限(output)
R1030  ; #1扭力下限(output)
R1032  ; #1扭力補償(output)
R1034  ; #1扭力上限+補償
R1036  ; #1扭力下限+補償
R1040  ; #2著座速度(set)
R1042  ; #2鎖緊速度(set)
R1044  ; #2著座扭力(set)
R1046  ; #2鎖緊扭力(set)
R1048  ; #2扭力上限(set)
R1050  ; #2扭力下限(set)
R1052  ; #2扭力補償(set)
R1060  ; #2著座速度(output)
R1062  ; #2鎖緊速度(output)
R1064  ; #2著座扭力(output)
R1066  ; #2鎖緊扭力(output)
R1068  ; #2扭力上限(output)
R1070  ; #2扭力下限(output)
R1072  ; #2扭力補償(output)
R1074  ; #2扭力上限+補償
R1076  ; #2扭力下限+補償
R1080  ; #3著座速度(set)
R1082  ; #3鎖緊速度(set)
R1084  ; #3著座扭力(set)
R1086  ; #3鎖緊扭力(set)
R1088  ; #3扭力上限(set)
R1090  ; #3扭力下限(set)
R1092  ; #3扭力補償(set)
R1100  ; #3著座速度(output)
R1102  ; #3鎖緊速度(output)
R1104  ; #3著座扭力(output)
R1106  ; #3鎖緊扭力(output)
R1108  ; #3扭力上限(output)
R1110  ; #3扭力下限(output)
R1112  ; #3扭力補償(output)
R1114  ; #3扭力上限+補償
R1116  ; #3扭力下限+補償
R1120  ; #4著座速度(set)
R1122  ; #4鎖緊速度(set)
R1124  ; #4著座扭力(set)
R1126  ; #4鎖緊扭力(set)
R1128  ; #4扭力上限(set)
R1130  ; #4扭力下限(set)
R1132  ; #4扭力補償(set)
R1140  ; #4著座速度(output)
R1142  ; #4鎖緊速度(output)
R1144  ; #4著座扭力(output)
R1146  ; #4鎖緊扭力(output)
R1148  ; #4扭力上限(output)
R1150  ; #4扭力下限(output)
R1152  ; #4扭力補償(output)
R1154  ; #4扭力上限+補償
R1156  ; #4扭力下限+補償
R1160  ; #5著座速度(set)
R1162  ; #5鎖緊速度(set)
R1164  ; #5著座扭力(set)
R1166  ; #5鎖緊扭力(set)
R1168  ; #5扭力上限(set)
R1170  ; #5扭力下限(set)
R1172  ; #5扭力補償(set)
R1180  ; #5著座速度(output)
R1182  ; #5鎖緊速度(output)
R1184  ; #5著座扭力(output)
R1186  ; #5鎖緊扭力(output)
R1188  ; #5扭力上限(output)
R1190  ; #5扭力下限(output)
R1192  ; #5扭力補償(output)
R1194  ; #5扭力上限+補償
R1196  ; #5扭力下限+補償
R1200  ; #6著座速度(set)
R1202  ; #6鎖緊速度(set)
R1204  ; #6著座扭力(set)
R1206  ; #6鎖緊扭力(set)
R1208  ; #6扭力上限(set)
R1210  ; #6扭力下限(set)
R1212  ; #6扭力補償(set)
R1220  ; #6著座速度(output)
R1222  ; #6鎖緊速度(output)
R1224  ; #6著座扭力(output)
R1226  ; #6鎖緊扭力(output)
R1228  ; #6扭力上限(output)
R1230  ; #6扭力下限(output)
R1232  ; #6扭力補償(output)
R1234  ; #6扭力上限+補償
R1236  ; #6扭力下限+補償
R1240  ; #7著座速度(set)
R1242  ; #7鎖緊速度(set)
R1244  ; #7著座扭力(set)
R1246  ; #7鎖緊扭力(set)
R1248  ; #7扭力上限(set)
R1250  ; #7扭力下限(set)
R1252  ; #7扭力補償(set)
R1260  ; #7著座速度(output)
R1262  ; #7鎖緊速度(output)
R1264  ; #7著座扭力(output)
R1266  ; #7鎖緊扭力(output)
R1268  ; #7扭力上限(output)
R1270  ; #7扭力下限(output)
R1272  ; #7扭力補償(output)
R1274  ; #7扭力上限+補償
R1276  ; #7扭力下限+補償
R1280  ; #8著座速度(set)
R1282  ; #8鎖緊速度(set)
R1284  ; #8著座扭力(set)
R1286  ; #8鎖緊扭力(set)
R1288  ; #8扭力上限(set)
R1290  ; #8扭力下限(set)
R1292  ; #8扭力補償(set)
R1300  ; #8著座速度(output)
R1302  ; #8鎖緊速度(output)
R1304  ; #8著座扭力(output)
R1306  ; #8鎖緊扭力(output)
R1308  ; #8扭力上限(output)
R1310  ; #8扭力下限(output)
R1312  ; #8扭力補償(output)
R1314  ; #8扭力上限+補償
R1316  ; #8扭力下限+補償
R1320  ; #9著座速度(set)
R1322  ; #9鎖緊速度(set)
R1324  ; #9著座扭力(set)
R1326  ; #9鎖緊扭力(set)
R1328  ; #9扭力上限(set)
R1330  ; #9扭力下限(set)
R1332  ; #9扭力補償(set)
R1340  ; #9著座速度(output)
R1342  ; #9鎖緊速度(output)
R1344  ; #9著座扭力(output)
R1346  ; #9鎖緊扭力(output)
R1348  ; #9扭力上限(output)
R1350  ; #9扭力下限(output)
R1352  ; #9扭力補償(output)
R1354  ; #9扭力上限+補償
R1356  ; #9扭力下限+補償
R1360  ; #10著座速度(set)
R1362  ; #10鎖緊速度(set)
R1364  ; #10著座扭力(set)
R1366  ; #10鎖緊扭力(set)
R1368  ; #10扭力上限(set)
R1370  ; #10扭力下限(set)
R1372  ; #10扭力補償(set)
R1380  ; #10著座速度(output)
R1382  ; #10鎖緊速度(output)
R1384  ; #10著座扭力(output)
R1386  ; #10鎖緊扭力(output)
R1388  ; #10扭力上限(output)
R1390  ; #10扭力下限(output)
R1392  ; #10扭力補償(output)
R1394  ; #10扭力上限+補償
R1396  ; #10扭力下限+補償
T2  ; 筒夾放鬆sol
T5  ; 夾緊氣缸放sol
